(* CoDeSys 2.3.9.1 project: oscat270.pro *)
(* Libraries: SysLibSockets.lib 14.4.05 11:11:38, WagoLibEthernet_01.lib 9.8.07 10:37:24, SysLibRtc.lib 5.10.04 09:37:42, Standard.lib 22.11.04 11:21:12, SYSLIBCALLBACK.LIB 20.4.05 10:04:48 *)

(* Global variable list: Constants *)
VAR_GLOBAL CONSTANT
	(* setup Parameters *)
	STEP7 : BOOL := FALSE;

	(* Mathematische Konstanten *)
	PI1 : REAL := 3.14159265358979323846264338327950288;	(* Kreiszahl PI *)
	PI2 : REAL := 6.283185307179586476;					(* PI * 2 *)
	E : REAL := 2.71828182845904523536028747135266249;	(* Eulersche Konstante *)

	(* Physikalische Konstanten *)
	C0 : REAL := 299792458 ;							(* Lichtgeschwindigkeit in m/s *)
	EL : REAL := 1.60217653E-19;						(* elementarladung in Colomb = A * s *)
	GN : REAL := 9.80665; 								(* Erdbeschleunigung in m / s² *)
	TK : REAL := -273.15;									(* absoluter Nullpunkt in °C *)
	RU : REAL := 8.314472; 								(*Universelle Gaskonstante in J / (mol · K) *)
	PN : REAL := 101325;									(* NormalDruck in Pa *)

END_VAR

VAR_GLOBAL
END_VAR

(* revisionhistory
hm 3.3.2007
	extended accuracy of pi2
	renamed T0 to Tk for better compatibility with other libraries
	renamed C t0 c0 for better compatibility

hm	2.5.2007
	added RU universal gas constant

hm	1. oct 2007
	added setup parameter STEP7

hm 31. oct 2007
	added PN
*)

(* Data type *)
TYPE esr_data :
STRUCT
	typ : BYTE;
	adress : STRING(10);
	DS : DT;
	TS : TIME;
	data : ARRAY[0..7] OF BYTE;
END_STRUCT
END_TYPE

(* Data type *)
TYPE vector_3 :
STRUCT
	X : REAL;
	Y : REAL;
	Z : REAL;
END_STRUCT
END_TYPE

(* POU XTEST/PLC_PRG, CFC *)
PROGRAM PLC_PRG
VAR
END_VAR
VAR_INPUT
END_VAR
_CFC_ (* Continuous Function Chart, elements in execution order *)
_END_CFC_
END_PROGRAM

(* POU XTEST/Baustein Tests/air_test, CFC *)
PROGRAM air_test
VAR
	temp: REAL := 70;
	den: REAL;
	den1: REAL;
	ent: REAL;
	cp: REAL;
	rh: REAL := 0.5;
	P: REAL := 101325;
	ice: BOOL;
	SDx: REAL;
	enth: REAL;
END_VAR
VAR (* helpers for the ST form of the networks *)
	_t1 : REAL;
	_t58 : REAL;
END_VAR
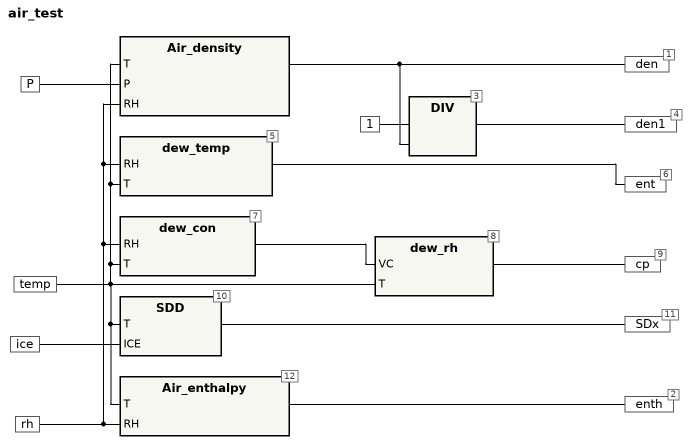
_CFC_ (* Continuous Function Chart, elements in execution order *)
#0 Air_density(T: temp, P: P, RH: rh)
#1 den <= #0
#2 enth <= #12
#3 DIV(1, #0)
#4 den1 <= #3
#5 dew_temp(RH: rh, T: temp)
#6 ent <= #5
#7 dew_con(RH: rh, T: temp)
#8 dew_rh(VC: #7, T: temp)
#9 cp <= #8
#10 SDD(T: temp, ICE: ice)
#11 SDx <= #10
#12 Air_enthalpy(T: temp, RH: rh)
_END_CFC_
(* the same logic as Structured Text *)
_t1 := Air_density(T := temp, P := P, RH := rh);
den := _t1;
enth := _t58;
den1 := 1 / _t1;
ent := dew_temp(RH := rh, T := temp);
cp := dew_rh(VC := dew_con(RH := rh, T := temp), T := temp);
SDx := SDD(T := temp, ICE := ice);
_t58 := Air_enthalpy(T := temp, RH := rh);
END_PROGRAM

(* POU mathematical/neg, ST *)
FUNCTION neg : INT
VAR_INPUT
	in : INT;
END_VAR
VAR
	X : WORD := 2#1111_1111_1111_1111;
END_VAR

(*
version 1.0	11 nov 2007
programmer 	hugo
tested by		tobias

this function return the value of in multiplied by -1

*)
neg := WORD_TO_INT(INT_TO_WORD(in - 1) XOR X);

(* revision history
hm 11.11.2007	rev 1.0
	original version

*)
END_FUNCTION

(* POU Building/HLK/Air_density, ST *)
FUNCTION Air_density : REAL
VAR_INPUT
	T : REAL;
	P : REAL;
	RH : REAL;
END_VAR
VAR CONSTANT
	RL : REAL := 287.05;
	RX : REAL := 3.773319E-3;
END_VAR
VAR
END_VAR

(*
version 1.1	4 dec 2007
programmer 	hugo
tested by		tobias

this function calculates the air density between 0 and 100 deg C

*)
Air_density := PN * (1 - RH * SDD(T, TRUE) * RX / P) / (RL * ( T - TK));

(* original code used for rev 1.0

SDD := SDD(T,FALSE);
RF := RL / (1- RH*SDD/P*RX);
Air_density := P / (RF * (T-TK));

*)

(* revision history

hm	29.10.2007		rev 1.0
	original version

hm	4.12.2007		rev 1.1
	changed code for better performance

*)
END_FUNCTION

(* POU Building/HLK/SDD, ST *)
FUNCTION SDD : REAL
VAR_INPUT
	T : REAL;
	ICE: BOOL;
END_VAR
VAR CONSTANT
END_VAR
VAR
END_VAR

(*
version 1.1	2 dec 2007
programmer 	hugo
tested by		tobias

this function calculates the vapor saturation pressure for moist Air over ice or water

*)
IF ice THEN
	SDD := 611.153 * EXP(22.4433 * T / (272.186 + T));
ELSE
	SDD := 611.213 * EXP(17.5043 * T / (241.2 + T));
END_IF;

(* old code used in rev 1.0
IF ice THEN
	SDD := 611.153 * exp10(9.747*T / (272.186 + T));
ELSE
	SDD := 611.213 * exp10(7.602*T / (241.2 + T));
END_IF;
*)


(* revision history

hm 29 oct 2007		rev 1.0
	original version

hm	2. dec 2007		rev 1.1
	changed code for better performance
*)
END_FUNCTION

(* POU Building/HLK/dew_temp, ST *)
FUNCTION dew_temp : REAL
VAR_INPUT
	RH : REAL;
	T : REAL;
END_VAR
VAR CONSTANT
	a : REAL := 7.5;
	b : REAL := 237.3;
END_VAR
VAR
	V : REAL;
END_VAR

(*
version 1.4	8 jan 2008
programmer 	hugo
tested by		tobias

this function calculates the dew point for air given the temperature and relative humidity.
dew_temp(60,0.25) = 16.7 °C.
which means the dew point for air with 25° and 60% RH is at 16.7 °C.


*)
IF rh > 0 THEN
(*	old code was rewritten for better performance
	SDD := 6.1078*EXPT(10,(a*T)/(b+T));
	DD := RH/100 * SDD;
	V := LOG(DD/6.1078);
	dew_temp := b*V/(a-v);
*)
	V := LOG(RH * 0.01 * exp10((a*T)/(b+T)));
	dew_temp := b*V/(a-V);
ELSE
	dew_temp:= -TK;
END_IF;

(* revision history

hm		2.10.2006	rev 1.0
	original version created

hm		29.4.2007	rev 1.1
	checked for rh not to be 0 because log(0) is not defined

hm		13.9.2007	rev 1.2
	code rewritten for better performance

hm		2. dec 2007	rev 1.3
	changed code for better performance

hm		8. jan 2008	rev 1.4
	further improvement in performance
*)

(*
Bezeichnungen:
r = relative Luftfeuchte
T = Temperatur in °C
TK = Temperatur in Kelvin (TK = T + 273.15)
TD = Taupunkttemperatur in °C
DD = Dampfdruck in hPa
SDD = Sättigungsdampfdruck in hPa

Parameter:
a = 7.5, b = 237.3 für T >= 0
a = 7.6, b = 240.7 für T < 0 über Wasser (Taupunkt)
a = 9.5, b = 265.5 für T < 0 über Eis (Frostpunkt)

R* = 8314.3 J/(kmol*K) (universelle Gaskonstante)
mw = 18.016 kg (Molekulargewicht des Wasserdampfes)
AF = absolute Feuchte in g Wasserdampf pro m3 Luft

Formeln:

   1. SDD(T) = 6.1078 * 10^((a*T)/(b+T))
   2. DD(r,T) = r/100 * SDD(T)
   3. r(T,TD) = 100 * SDD(TD) / SDD(T)
   4. TD(r,T) = b*v/(a-v) mit v(r,T) = log10(DD(r,T)/6.1078)
   5. AF(r,TK) = 10^5 * mw/R* * DD(r,T)/TK; AF(TD,TK) = 10^5 * mw/R* * SDD(TD)/TK 

*)
END_FUNCTION

(* POU mathematical/exp10, ST *)
FUNCTION exp10 : REAL
VAR_INPUT
	X : REAL;
END_VAR
VAR
END_VAR

(*
version 1.0	 2 dec 2007
programmer 	hugo
tested by		tobias

this function calculates the exponent to the basis 10
exp10(3) = 1000

*)
exp10 := EXP(X * 2.30258509299405);

(* revision history
hm	2. dec 2007		rev 1.0
	original version

*)
END_FUNCTION

(* POU Building/HLK/dew_con, ST *)
FUNCTION dew_con : REAL
VAR_INPUT
	RH : REAL;
	T : REAL;
END_VAR
VAR CONSTANT
END_VAR
VAR
END_VAR

(*
version 1.2	2 dec 2007
programmer 	hugo
tested by		tobias

this function calculates the water concentratin in air for a given temperature and relative humidity.
the output states the concentration of water vapor in air in Gramms / qubic meter.

*)
IF rh > 0 THEN
(*	this code is good to read but need to be improoved
	SDD := 6.1078*EXPT(10,(a*T)/(b+T));
	DD := RH/100 * SDD;
	V := LOG(DD/6.1078);
	TD := b*V/(a-v);
	dew_con := 0.1 * mw / RU * DD / (T - TK);
*)
	dew_con := 2.166824303E-2 * RH * SDD(T,FALSE)  / (T - TK);
ELSE
	dew_con := 0;
END_IF;

(*
Bezeichnungen:
r = relative Luftfeuchte
T = Temperatur in °C
TK = Temperatur in Kelvin (TK = T + 273.15)
TD = Taupunkttemperatur in °C
DD = Dampfdruck in hPa
SDD = Sättigungsdampfdruck in hPa

Parameter:
a = 7.5, b = 237.3 für T >= 0
a = 7.6, b = 240.7 für T < 0 über Wasser (Taupunkt)
a = 9.5, b = 265.5 für T < 0 über Eis (Frostpunkt)

R* = 8314.3 J/(kmol*K) (universelle Gaskonstante)
mw = 18.016 kg (Molekulargewicht des Wasserdampfes)
AF = absolute Feuchte in g Wasserdampf pro m3 Luft

Formeln:

   1. SDD(T) = 6.1078 * 10^((a*T)/(b+T))
   2. DD(r,T) = r/100 * SDD(T)
   3. r(T,TD) = 100 * SDD(TD) / SDD(T)
   4. TD(r,T) = b*v/(a-v) mit v(r,T) = log10(DD(r,T)/6.1078)
   5. AF(r,TK) = 10^5 * mw/R* * DD(r,T)/TK; AF(TD,TK) = 10^5 * mw/R* * SDD(TD)/TK 

*)

(* revision history

hm 29 apr 2007		rev 1.0
	original version

hm	13.sep 2007		rev 1.1
	improoved coding for speed
	deleted unused variabled SDD,DD,V, TD

hm	2. dec 2007		rev 1.2
	changed code for better performance
	output is now in Gramms / Qubic meter
*)
END_FUNCTION

(* POU Building/HLK/dew_rh, ST *)
FUNCTION dew_rh : REAL
VAR_INPUT
	VC : REAL;
	T : REAL;
END_VAR

(*
version 1.1	2 dec 2007
programmer 	hugo
tested by		tobias

this function calculates the relative humidity in air for a given temperature in °C and vapor concentration in Kg/m³..

*)
dew_rh := LIMIT(0,VC / dew_con(1,T),100);

(* code before rev 1.1
dew_rh := VC / dew_con(100,T) * 100;
IF dew_rh > 100 THEN dew_rh := 100; END_IF;
*)

(* revision history
hm		29. apr 2007	rev 1.0
	original version

hm		2. 12. 2007		rev 1.1
	new code for better performance

*)
END_FUNCTION

(* POU Building/HLK/Air_enthalpy, ST *)
FUNCTION Air_enthalpy : REAL
VAR_INPUT
	T : REAL;
	RH : REAL;
END_VAR
VAR CONSTANT
	CPL : REAL := 1.00482;
	CW : REAL := 1.86;
	LH : REAL := 2500.78;
END_VAR
VAR
END_VAR

(*
version 1.1	2 nov 2007
programmer 	hugo
tested by		tobias

this function calculates the enthalpy for humid air between 0 and 100 deg C

*)
Air_enthalpy := CPL * T + (CW * T + LH) * dew_con(RH,T);

(* revision history

hm	31.10.2007		rev 1.0
	original version

hm	2.11.2007		rev 1.1
	deleted unused variable RF

hm	2.12.2007		rev 1.2
	changed code for better performance
*)
END_FUNCTION

(* POU XTEST/Baustein Tests/bcd_test, CFC *)
PROGRAM bcd_test
VAR
	strbcd: STRING;
	inout: INT;
	inx: INT;
END_VAR
VAR_INPUT

END_VAR
VAR (* helpers for the ST form of the networks *)
	_t16 : BCD;
	_t15 : INT;
END_VAR
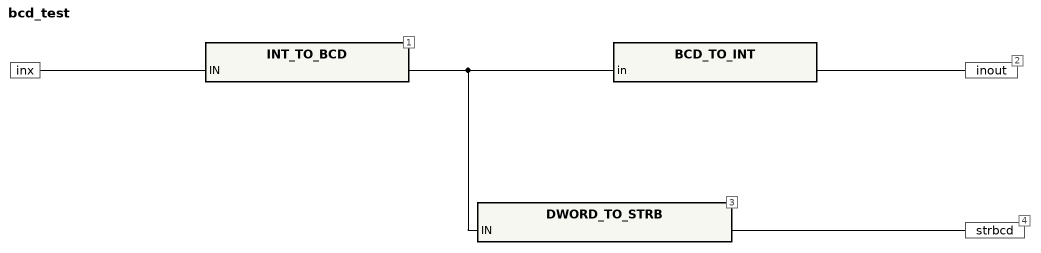
_CFC_ (* Continuous Function Chart, elements in execution order *)
#0 BCD_TO_INT(in: #1)
#1 INT_TO_BCD(IN: inx)
#2 inout <= #0
#3 DWORD_TO_STRB(IN: #1)
#4 strbcd <= #3
_END_CFC_
(* the same logic as Structured Text *)
_t15 := BCD_TO_INT(in := _t16);
_t16 := INT_TO_BCD(IN := inx);
inout := _t15;
strbcd := DWORD_TO_STRB(IN := _t16);
END_PROGRAM

(* POU Logic/gate logic/BCD_TO_INT, ST *)
FUNCTION BCD_TO_INT : INT
VAR_INPUT
	in : BYTE;
END_VAR
VAR
END_VAR

(*
version 1.0	13 dec 2007
programmer 	hugo
tested by		tobias

this function converts a two digit bcd number into an integer.
*)
	BCD_TO_INT := (in AND 16#0F) + (SHR(in,4) * 10);

(* revision history
hm	13.12.2007
	original version

*)
END_FUNCTION

(* POU Logic/gate logic/INT_TO_BCD, ST *)
FUNCTION INT_TO_BCD : BYTE
VAR_INPUT
	IN : INT;
END_VAR
VAR
END_VAR

(*
version 1.0	17 jan 2007
programmer 	hugo
tested by		tobias

this function converts an integer into a two digit bcd number.
*)
INT_TO_BCD := INT_TO_BYTE(SHL(TRUNC(in/10),4) + (in MOD 10));

(* revision history
hm	13.12.2007
	original version

*)
END_FUNCTION

(* POU String/DWORD_TO_STRB, ST *)
FUNCTION DWORD_TO_STRB : STRING
VAR_INPUT
	IN : DWORD;
END_VAR
VAR
	pt : POINTER TO BYTE;
	i: INT;
END_VAR

(*
version 1.1	15 dec 2007
programmer 	hugo
tested by		tobias

DWORD_TO_STRINGB converts a DWORD to a String of Bits represented by '0' and '1' s.
The lowest order bit will be on the right and the high order bit on the left.

*)
(* pointer für die ausgabe ermitteln *)
pt := ADR(DWORD_TO_STRB);
(* die 8 ausgabecharacter ermitteln und schreiben *)
FOR i := 1 TO 32 DO
	IF in.31 THEN pt^ := 49; ELSE pt^ := 48; END_IF;
	in := SHL(in,1);
	pt := pt + 1;
END_FOR;

(* der ausgabestring muss nochg mit 0 abgeschlossen werden *)
pt^ := 0;

(* revision history
hm		9.6.2007	rev 1.0		
	original version 
hm		15.dec 2007	rev 1.1
	changed code for better performance
*)
END_FUNCTION

(* POU XTEST/Baustein Tests/blind_test, CFC *)
PROGRAM blind_test
VAR
	up: BOOL;
	dn: BOOL;
	x1: blind_scene;
	mu: BOOL;
	md: BOOL;
	pos: BYTE;
	ang: BYTE;
	x2: blind_security;
	esr: BYTE;
	fire: BOOL;
	wind: BOOL;
	alarm: BOOL;
	rain: BOOL;
	x3: blind_control;
	x5: blind_input;
	p: BYTE;
	a: BYTE;
	IN: BOOL;
	utc: DT;
	X7: blind_night;
	x8: sun_time;
	Door: BOOL;
	x9: sun_pos;
	x10: BLIND_SHADE;
	S_write: BOOL;
	S_enable: BOOL;
	scene: BYTE;
	sun: BOOL;
	ex: BOOL;
END_VAR
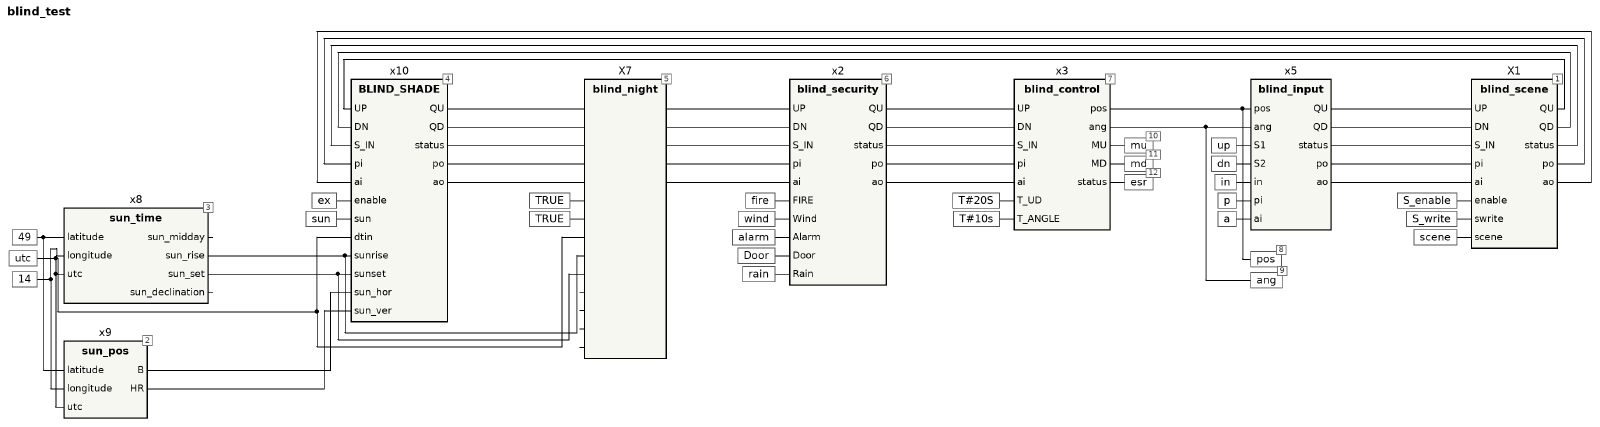
_CFC_ (* Continuous Function Chart, elements in execution order *)
#0 x5:blind_input(pos: #7.pos, ang: #7.ang, S1: up, S2: dn, in: in, pi: p, ai: a, click_mode := TRUE, click_time := T#250ms, manual_timeout := T#10s)
#1 X1:blind_scene(UP: #0.QU, DN: #0.QD, S_IN: #0.status, pi: #0.po, ai: #0.ao, enable: S_enable, swrite: S_write, scene: scene)
#2 x9:sun_pos(latitude: 49, longitude: 14, utc: utc)
#3 x8:sun_time(latitude: 49, longitude: 14, utc: utc)
#4 x10:BLIND_SHADE(UP: #1.QU, DN: #1.QD, S_IN: #1.status, pi: #1.po, ai: #1.ao, enable: ex, sun: sun, dtin: utc, sunrise: #3.sun_rise, sunset: #3.sun_set, sun_hor: #2.B, sun_ver: #2.HR, direction := 180, slat_width := 60, Slat_spacing := 60)
#5 X7:blind_night(#4.QU, #4.QD, #4.status, #4.po, #4.ao, TRUE, TRUE, utc, #3.sun_rise, #3.sun_set, -, -, -, -)
#6 x2:blind_security(UP: #5.out 1, DN: #5.out 2, S_IN: #5.out 3, pi: #5.out 4, ai: #5.out 5, FIRE: fire, Wind: wind, Alarm: alarm, Door: Door, Rain: rain, Alarm_UP := TRUE)
#7 x3:blind_control(UP: #6.QU, DN: #6.QD, S_IN: #6.status, pi: #6.po, ai: #6.ao, T_UD: T#20S, T_ANGLE: T#10s, sens := 5, T_Lockout := T#3s)
#8 pos <= #7.pos
#9 ang <= #7.ang
#10 mu <= #7.MU
#11 md <= #7.MD
#12 esr <= #7.status
_END_CFC_
END_PROGRAM

(* POU Building/Jalousie/blind_scene, ST *)
FUNCTION_BLOCK blind_scene
VAR_INPUT
	UP, DN : BOOL;
	S_IN : BYTE;
	pi, ai : BYTE;
	enable : BOOL;
	swrite : BOOL;
	scene : BYTE;
END_VAR
VAR_INPUT CONSTANT
END_VAR
VAR_OUTPUT
	QU, QD : BOOL;
	status : BYTE;
	po, ao : BYTE;
END_VAR
VAR RETAIN
	sx : ARRAY[0..15,0..2] OF BYTE;
END_VAR
VAR_TEMP
	x : BYTE;

END_VAR

(*
version 1.1	29. jan 2008
programmer 	hugo
tested by		tobias


*)
(* delete all bits except the lower 4 of scene *)
x := scene AND 16#0F;

IF enable AND sx[x,2] > 0 AND UP AND DN THEN
	po := sx[x,0];
	ao := sx[x,1];
	status := 160 + x;  (* Status number is 160 to 175 for the 16 scenes *)
	QU := TRUE;
	QD := TRUE;
ELSE
	QU := UP;
	QD := DN;
	status := S_IN;
	po := pi;
	ao := ai;
END_IF;

(* write scene if necessary *)
IF swrite THEN
	status := 176;		(* write scene *)
	sx[x,0] := pi;
	sx[x,1] := ai;
	IF enable THEN sx[x,2] := 1; ELSE sx[x,2] := 0; END_IF; (* if sx[x,2] = 0 the scene is disabled *)
END_IF;


(* revision history
hm	24. oct 2007	rev 1.0
	original release

hm		29.1.2008	rev 1.1
	replaced shr/shl with and for better performance
*)
END_FUNCTION_BLOCK

(* POU Building/Jalousie/blind_security, ST *)
FUNCTION_BLOCK blind_security
VAR_INPUT
	UP, DN : BOOL;
	S_IN : BYTE;
	pi, ai : BYTE;
	FIRE : BOOL;
	Wind : BOOL;
	Alarm : BOOL;
	Door : BOOL;
	Rain : BOOL;
END_VAR
VAR_INPUT CONSTANT
	Alarm_UP : BOOL := TRUE;
END_VAR
VAR_OUTPUT
	QU, QD : BOOL;
	status : BYTE;
	po, ao : BYTE;
END_VAR
VAR
END_VAR

(*
version 1.1	6. oct 2007
programmer 	hugo
tested by		tobias


*)
IF Fire THEN
	QU := TRUE;
	QD := FALSE;
	status := 111;
ELSIF Wind THEN
	QU := TRUE;
	QD := FALSE;
	status := 112;
ELSIF alarm THEN
	QU := Alarm_up;
	QD := NOT Alarm_up;
	status := 113;
ELSIF Door THEN
	QU := TRUE;
	QD := FALSE;
	status := 114;
ELSIF Rain AND NOT (up XOR dn) THEN
	QU := FALSE;
	QD := TRUE;
	status := 115;
ELSE
	QU := UP;
	QD := DN;
	status := S_IN;
	po := pi;
	ao := ai;
END_IF;


(* revision history
hm	29. sep 2007	rev 1.0
	original release

hm	6. oct 2007		rev 1.1
	added pos and angle inputs and outputs
	manual will override rain position
	alarm position can now be configured

*)
END_FUNCTION_BLOCK

(* POU Building/Jalousie/blind_control, ST *)
FUNCTION_BLOCK blind_control
VAR_INPUT
	UP, DN : BOOL;
	S_IN : BYTE;
	pi : BYTE;
	ai : BYTE;
	T_UD, T_ANGLE : TIME;
END_VAR
VAR_INPUT CONSTANT
	sens : BYTE := 5;
	T_Lockout: TIME := T#100ms;
END_VAR
VAR_OUTPUT
	pos, ang : BYTE;
	MU, MD : BOOL;
	status : BYTE;
END_VAR
VAR
	act : blind_actuator;
	delta : BYTE;
END_VAR

(*
version 1.3	30. oct 2007
programmer 	hugo
tested by		tobias


*)
IF UP AND DN THEN
	(* automatic modus detected *)
	(* first find correct position *)
	IF BYTE_TO_INT(act.pos) < BYTE_TO_INT(pi) - delta THEN
		act.UP := TRUE;
		act.DN := FALSE;
		delta := 0;
		act.S_IN := 121;
	ELSIF BYTE_TO_INT(act.pos) > BYTE_TO_INT(pi) + delta THEN
		act.UP := FALSE;
		act.DN := TRUE;
		delta := 0;
		act.S_IN := 122;
	(* regulate angle *)
	ELSIF BYTE_TO_INT(act.ang) < BYTE_TO_INT(ai) - delta AND T_angle > T#100ms THEN
		act.UP := TRUE;
		act.DN := FALSE;
		delta := 0;
		act.S_IN := 123;
	ELSIF BYTE_TO_INT(act.ang) > BYTE_TO_INT(ai) + delta AND T_angle > T#100ms THEN
		act.UP := FALSE;
		act.DN := TRUE;
		delta := 0;
		act.S_IN := 124;
	(* correct position reached *)
	ELSE
		act.UP := FALSE;
		act.DN := FALSE;
		delta := sens;
		act.S_IN := 0;
	END_IF;
ELSE
	act.UP := UP;
	act.DN := DN;
END_IF;

(* hand over status *)
IF s_in > 0 THEN act.S_IN := S_IN; END_IF;

(* blind control calls blind_actuator *)
act(T_UD:=T_UD, T_ANGLE:=T_ANGLE, T_lockout := T_Lockout);
pos := act.pos;
ang := act.ang;
MU := act.QU;
md := act.QD;
status := act.status;

(* revision history
hm	29. sep 2007	rev 1.0
	original release

hm	6. oct 2007		rev 1.1
	rearranged outputs
	integrated blind_actuator into blind_control

hm	16. oct 2007	rev 1.2
	ignore angle when t_angle = 0

hm 29. oct 2007	rev 1.3
	added lockout configuration time for motor direction change
	sens has a setup value of 5
*)
END_FUNCTION_BLOCK

(* POU Building/Jalousie/blind_actuator, ST *)
 FUNCTION_BLOCK blind_actuator
VAR_INPUT
	UP, DN : BOOL;
	S_IN : BYTE;
	T_UD : TIME := T#10s;
	T_Angle : TIME := T#3s;
END_VAR
VAR_INPUT CONSTANT
	T_lockout : TIME := t#100ms;
END_VAR
VAR_OUTPUT
	pos, ang : BYTE;
	QU, QD : BOOL;
	status : BYTE;
END_VAR
VAR
	position, angle : rmp_B;
	lock : interlock;
END_VAR

(*
version 1.1	6 oct 2007
programmer 	hugo
tested by		tobias

blind actuator drives the up and down motor of a blind. T_lockout specifies the time between up or dn becomes active. 
To change direction there must be a minimum wait time to allow the motors to come to rest first.
the up and down outputs QU and QD are controlled by the inputs UP and DN.
the outputs pos and ang simulate the position of the blind pos = 0 means blind is down and pos = 255 = blind is up.
the angle 0 means vertical posisition of the slates and 255 means horizontal position of the slates.


*)
(* make sure only one motor is active at a given time *)
lock(i1 := UP, I2 := DN, TL := T_lockout);

(* ramp up or down to simulate the angle position of the blind slats *)
angle(en := lock.Q1 OR lock.Q2, UP := lock.Q1, PT := T_Angle);
position(en := lock.Q1 AND angle.high OR lock.Q2 AND angle.low, up := lock.Q1, PT := T_UD);

(* set the outputs *)
pos := position.Out;
ang := angle.Out;
QU := lock.Q1;
QD := lock.Q2;

(* set the status output *)
IF UP AND DN THEN
	IF s_in < 10 AND S_in > 1 THEN status := s_in; ELSE status := 1; END_IF;			(* error up and down together are not allowed *)
ELSIF S_IN > 0 THEN
	status := S_IN;
ELSIF UP THEN
	status := 101;
ELSIF DN THEN
	status := 102;
ELSE
	status := 0;
END_IF;


(* revision history
hm	29. sep 2007	rev 1.0
	original release

hm	6. oct 2007		rev 1.1
	rearranged outputs
	
*)
END_FUNCTION_BLOCK

(* POU engineering/signal generators/rmp_B, ST *)
FUNCTION_BLOCK rmp_B
VAR_INPUT
	SET : BOOL := FALSE;
	PT : TIME;
	EN : BOOL := TRUE;
	UP : BOOL := TRUE;
	RST : BOOL := FALSE;
END_VAR
VAR_OUTPUT
	out : BYTE;
	busy: BOOL;
	high : BOOL;
	low : BOOL;
END_VAR
VAR
	last_step : DWORD;
	now : DWORD;
	tmp: DWORD;
	edge: BOOL;
	N : BYTE;
	init: BOOL;
END_VAR

(*
	version 1.6	25 dec 2007
	programmer 	oscat
	tested BY		oscat

this ramp generator generates a byte wide ramp with 255 steps
the generator has an asynchronous set and reset
the ramp is controlled by PT which is the total ramp time for a full sweep from 0..255
an UD input controlls the direction Up or Down and the E input enables the ramp generation
a busy output indicates that the ramp is running, busy false means output is stable.
the outputs low and high will be true when the output has reached its max or min value.

*)
(* read system time *)
now := T_PLC_MS();

(* init code for startup *)
IF NOT init THEN
	init := TRUE;
	last_step := now;
END_IF;

(* calculate the necessary step response *)
IF pt = t#0s THEN
	tmp := 255;
ELSE
	tmp := SHL(now - last_step, 8) / (TIME_TO_DWORD(pt));
END_IF;
IF tmp > 255 THEN N:= 255; ELSE N:= DWORD_TO_BYTE(tmp); END_IF;

(* detetct edge on en *)
IF en AND NOT edge THEN
	last_step := now;
(* check for asynchronous set or reset *)
ELSIF rst THEN
	out := 0;
ELSIF set  THEN
	out := 255;
ELSIF en AND N > 0 THEN
	(* generate ramp *)
	last_step := now;
	IF UP THEN
		IF out > 255 - N THEN out := 255; ELSE out := out + N; END_IF;
	ELSE
		IF out < N THEN out := 0; ELSE out := out - N; END_IF;
	END_IF;
END_IF;
edge := en;

(* checks for outputs stable and reset or set busy flag *)
IF out = 0 THEN
	busy := FALSE;
	low := TRUE;
	high := FALSE;
ELSIF out = 255 THEN
	busy := FALSE;
	high := TRUE;
	low := FALSE;
ELSE
	busy := en;
	high := FALSE;
	low := FALSE;
END_IF;


(* revision history

hm 5.10.2006	rev 1.1
	added busy output
hm 17.1.2007	rev 1.2
	renamed input ud to up for better usability
	deleted unused variable step

hm	17.9.2007	rev 1.3
	replaced time() with t_plc_ms() for compatibility reasons

hm	28. sep 2007	rev 1.4
	added outputs on and off
	busy is now disabled while en is false
	new coding for higher accuracy and performance

hm	5. oct 2007		rev 1.5
	added statements to allow for PT to be t#0s output jumps to max or min immediately

hm	25. dec 2007	REV 1.6
	IMPROOVED CODE FOR BETTER PERFORMANCE
*)
END_FUNCTION_BLOCK

(* POU engineering/measurements/T_PLC_MS, ST *)
FUNCTION T_PLC_MS : DWORD
VAR CONSTANT
	debug : BOOL := FALSE;
	N : INT := 0;
	offset : DWORD := 0;
END_VAR
VAR
	tx : TIME;
	temp : DWORD := 1;
END_VAR

(*
version 1.1	12 nov 2007
programmer 	hugo
tested by		tobias

T_PLC_MS reads the internal PLC timer and return the time, it has the advantage to be able to set a debug mode 
and speed up the counter to test the plc timer overrun which occurs every 50 days respectively 25 days at siemens S7
this routine also allows to correct the behavior of s7 where the internal plc counter will not count all 32 bits.

*)
tx := TIME();
T_PLC_MS := TIME_TO_DWORD(Tx);
(* hier muss die korrektur für step7 stattfinden
plctime muss den vollen wertebereich von time ausnutzen:
wenn bei step7 time -24tage bis plus 24 tage ist dann muss der timer auch beim überlauf auf -24tage springen 
und auf keinen fall auf 0 !!!!
für siemens muss ein weiterer fb im main eingebunden werden der sicherstellt das alle 32 bits durchgezählt werden.
es kann nur ein fb sein den er muss sich das oberste (32te) bit merken.
oder etwa spring s7 bei überlauf auf -24 tage????? dann wäre keine korrektur nötig.
*)
IF debug THEN
	T_PLC_MS := (SHL(T_PLC_MS,N) OR SHL(temp,N)-1) + Offset;
END_IF;

(* revision history
hm	14.9.2007	rev 1.0
	original version

hm	12. nov 2007	rev 1.1
	added temporaray variable tx because some compilers could not handle time() as an argument

*)
END_FUNCTION

(* POU engineering/signal processing/Offset, ST *)
FUNCTION Offset : REAL
VAR_INPUT
	X : REAL;
	O1, O2, O3, O4 : BOOL;
	D : BOOL;
END_VAR
VAR_INPUT CONSTANT
	Offset_1 : REAL;
	Offset_2 : REAL;
	Offset_3 : REAL;
	Offset_4 : REAL;
	default : REAL;
END_VAR

(*
version 1.0	12 jan 2007
programmer 	oscat
tested by		tobias

The Function offset adds offsets to an analog signal depending on digital inputs.
all selected offsets are added at the same time.
with the input D a default value instead of the input X can be used.

*) 
IF D THEN Offset := default; ELSE Offset := X; END_IF;
IF O1 THEN Offset := Offset + offset_1; END_IF;
IF O2 THEN Offset := Offset + offset_2; END_IF;
IF O3 THEN Offset := Offset + offset_3; END_IF;
IF O4 THEN Offset := Offset + offset_4; END_IF;
END_FUNCTION

(* POU engineering/automation/interlock, ST *)
FUNCTION_BLOCK interlock
VAR_INPUT
	I1, I2 : BOOL;
	TL : TIME;
END_VAR
VAR_OUTPUT
	Q1, Q2 : BOOL;
END_VAR
VAR
	T1, T2 : TOF;
END_VAR

(*
version 1.0	28 sep 2007
programmer 	hugo
tested by		tobias

INTERLOCK has two inputs I1 and I2 which drive the corresponding outputs Q1 and Q2.
the inputs signals lock each other out and therfore I1 can only drive Q1 when I2 is Low and vice versa.
The input TL specifies a dead time between two outputs can become active.
an output can only become active when the other output was not active for the time TL.

*)
(* the input signal have a run delay to lockout the other input *)
T1(IN := I1, PT := TL);
T2(IN := I2, PT := TL);

Q1 := I1 AND NOT t2.Q;
Q2 := I2 AND NOT t1.Q;


(* revision history

hm	28 sep 2007		rev 1.0
	original version

*)
END_FUNCTION_BLOCK

(* POU Building/Jalousie/blind_input, ST *)
FUNCTION_BLOCK blind_input
VAR_INPUT
	pos, ang : BYTE;
	S1, S2 : BOOL;
	in : BOOL;
	pi, ai : BYTE;
END_VAR
VAR_INPUT CONSTANT
	single_switch : BOOL := FALSE;
	click_mode : BOOL := TRUE;
	click_time : TIME := T#200ms;
	click_timeout : TIME := T#60s;
	manual_timeout: TIME := T#1h;
END_VAR
VAR_OUTPUT
	QU, QD : BOOL;
	status : BYTE;
	po, ao : BYTE;
END_VAR
VAR
	click_run : TOF;
	tog1, tog2 : TOGGLE;
	pl1, pl2 : Pulse_Length;
	SU, SD : BOOL;
	last_act: DWORD;
	tx: DWORD;
END_VAR

(*
version 1.2	30 dec 2007
programmer 	hugo
tested by		tobias


*)
(* read system_time *)
tx := T_PLC_MS();

(* single or double switch operation *)
IF click_mode THEN
	PL1(in := S1, T_short := click_time, T_long := click_time);
	PL2(in := S2, T_short := click_time, T_long := click_time);
	(* a timeout needs to be added for click enable *)
	click_run(IN := pl1.short OR pl2.short, PT := click_timeout);
	tog1(clk := pl1.short, rst := pl1.long OR pl2.short OR pl2.long OR NOT click_run.Q);
	tog2(clk := pl2.short, rst := pl2.long OR pl1.short OR pl1.long OR NOT click_run.Q);

	SU := tog1.Q OR PL1.long;
	SD := tog2.Q OR pl2.long;
ELSE
	tog1(CLK := NOT S1);
	SU := (S1 AND NOT tog1.Q AND single_switch) OR (NOT single_switch AND S1);
	SD := (S1 AND tog1.Q AND single_switch) OR (NOT single_switch AND S2);
END_IF;

(* Forced Input is active *)
IF in THEN
	QU := TRUE;
	QD := TRUE;
	po := pi;
	ao := ai;
	status := 131;

(* in manual mode set ps and as to actual values *)
ELSIF SU OR SD THEN
	po := pos;
	ao := ang;
	last_act := tx;
	QU := SU;
	QD := SD;
	IF su THEN status := 132; ELSE status := 133; END_IF;

(* enable automatik mode after auto timer has expired *)
ELSIF manual_timeout > t#0s AND tx - last_act >= TIME_TO_DWORD(manual_timeout) THEN
	QU := TRUE;
	QD := TRUE;
	status := 134;

(* no input active *)
ELSE
	QU := FALSE;
	QD := FALSE;
	status := 0;
END_IF;


(* revision history
hm	29. sep 2007	rev 1.0
	original release

hm	6. oct 2007		rev 1.1
	renamed ps and as to po and ao

hm	30. dec 2007	rev 1.2
	added click_timeout variable and function

*)
END_FUNCTION_BLOCK

(* POU Logic/FF edge triggered/TOGGLE, ST *)
FUNCTION_BLOCK TOGGLE
VAR_INPUT
	CLK : BOOL;
	rst : BOOL := FALSE;
END_VAR
VAR_OUTPUT
	Q : BOOL;
END_VAR
VAR
	edge : BOOL;
END_VAR

(*
version 1.0	13 sep 2007
programmer 	hugo
tested by		tobias

toggle flip flop the output changes state with every rising edge of clk.

*)
IF rst THEN
	q := 0;
ELSIF clk AND NOT edge THEN
	Q := NOT Q;
END_IF;
edge := clk;

(* revision history

hm	13.9.2007		rev 1.0
	original version

*)
END_FUNCTION_BLOCK

(* POU Building/electrical/Pulse_Length, ST *)
FUNCTION_BLOCK Pulse_Length
VAR_INPUT
	in : BOOL;
END_VAR
VAR_OUTPUT
	short : BOOL;
	middle : BOOL;
	long : BOOL;
END_VAR
VAR_INPUT CONSTANT
	T_short : TIME := t#100ms;
	T_long : TIME := t#1s;
END_VAR
VAR
	tx : TIME;
	tn: TIME;
	edge : BOOL;
END_VAR

(*
version 1.1	15 sep 2007
programmer 	oscat
tested by		tobias

Pulse_length indicates on 3 outputs if an input pulse had been shorter than T_short (short = True), longer than T_long (long = True) or between T_short and T_long (middle = True).

*)
(* read system time *)
tx := DWORD_TO_TIME(T_PLC_MS());

(* reset outputs, they should only be active 1 cycle *)
short := FALSE;
Middle := FALSE;
long := FALSE;

(* detect rising edge *)
IF in AND NOT edge THEN
	edge := TRUE;
	tn := tx;

(* detect for falling edge *)
ELSIF NOT in AND edge THEN
	edge := FALSE;
	tn := tx - tn;
	IF tn < t_short THEN
		short := TRUE;
	ELSIF tn > t_long THEN
		long := TRUE;
	ELSE
		Middle := TRUE;
	END_IF;

(* generate long pulse as soon as T_long is reached *)
ELSIF in AND tx - tn > t_long THEN
	long := TRUE;
END_IF;


(* revision history

hm	15. feb 2006	rev 1.0
	original version

hm	15 sep 2007		rev 1.1
	replaced Time() with T_PLC_MS for compatibility and performance reasons

*)
END_FUNCTION_BLOCK

(* POU Building/Jalousie/blind_night, ST *)
FUNCTION_BLOCK blind_night
VAR_INPUT
	UP, DN : BOOL;
	S_IN : BYTE;
	pi, ai : BYTE;
	E_night : BOOL := TRUE;
	E_day	: BOOL := TRUE;
	dtin : DT;
	sunrise, sunset : TOD;
END_VAR
VAR_INPUT CONSTANT
	sunrise_offset : TIME;
	sunset_offset : TIME;
	night_position : BYTE := 0;
	night_angle : BYTE := 0;
END_VAR
VAR_OUTPUT
	QU, QD : BOOL;
	status : BYTE;
	po, ao : BYTE;
END_VAR
VAR
	night : BOOL;
	last_night, last_day : DATE;
END_VAR

(*
version 1.2	6 oct 2007
programmer 	hugo
tested by		tobias


*)
IF NOT (up AND dn) AND night THEN
	(* manual operation at night will cancel operation for one night *)
	night := FALSE;
ELSIF (DT_TO_TOD(dtin) > sunset + sunset_offset) AND (last_night < DT_TO_DATE(dtin)) AND NOT night AND e_night THEN
	(* enable night *)
	night := TRUE;
	last_night := DT_TO_DATE(dtin);
ELSIF (DT_TO_TOD(dtin) > sunrise + sunrise_offset) AND (last_day < DT_TO_DATE(dtin)) AND night AND e_day AND (last_night < DT_TO_DATE(dtin)) THEN
	(* disable night *)
	night := FALSE;
	last_day := DT_TO_DATE(dtin);
END_IF;

(* shade at night only in auto mode and enable = true *)
IF UP AND DN AND night THEN
	status := 141;
	po := night_position;
	ao := night_angle;
ELSE
	QU := UP;
	QD := DN;
	po := pi;
	ao := ai;
	status := s_in;
END_IF;


(* revision history
hm	29. sep 2007	rev 1.0
	original version

hm	5. oct 2007		rev 1.1
	added enable input

hm	6. oct 2007		rev 1.2
	added pos and angle inputs and outputs
	night position and angle can now be configured
	any manual operation at night will cancel night operation

*)
END_FUNCTION_BLOCK

(* POU Time&Date/sun_time, ST *)
FUNCTION_BLOCK sun_time
VAR_INPUT
	latitude : REAL;				(* latitude of geographical position  *)
	longitude : REAL;				(* longitude of geographical position  *)
	utc : DT;						(*	world time				*)
END_VAR
VAR_OUTPUT
	sun_midday : TOD;			(*	astrological midday in hours when sun stand at south direction	*)
	sun_rise : TOD;				(*	sun rise for current day in local time *)
	sun_set : TOD;				(*	sun set for current day in local time *)
	sun_declination : REAL;		(*	sun declination at midday in degrees	*)
END_VAR
VAR
	T: INT;							(* day in the year   *)
	DK: REAL;						(* sun declination at midday *)
	delta: REAL;					(* delta from midday for sunrise and sunset  *)
	h: REAL;
	B: REAL;
	offset : REAL;
	l15: REAL;
	dat: DATE;
	last_dat: DATE;
END_VAR

(*
version 1.4	17. jan 2008
programmer 	hugo
tested by		tobias

this FUNCTION block calculates the sun rise, sun set, sun offset at midday sun declination for a given date 
for performance reasons the algorithm has been simplified and is accurate within a few minutes only 
the times are calculated in utc and have to be corrected for the given time zone
this correction is not done within sun_time because it would be a problem on days where dst is enabled or disabled


*)
dat := DT_TO_DATE(utc);
IF dat = last_dat THEN RETURN; END_IF;
last_dat := dat;
l15 := longitude * 0.0666666666666;
B := latitude * 0.0174532925199433;
h := -0.0145;
T := day_of_year(dat);
offset := -0.1752 * SIN(0.033430*T + 0.5474) - 0.1340*SIN(0.018234*T - 0.1939);
sun_midday := hour_to_tod(12 + Offset - l15);
DK := 0.40954 * SIN(0.0172 * (T-79.35));
sun_declination := deg(DK);
delta := 12*ACOS((SIN(h) - SIN(B) * SIN(DK)) / (COS(B) * COS(DK))) * 0.318309886;
sun_rise := hour_to_tod(12 - delta - Offset - l15);
sun_set := hour_to_tod(12 + delta - Offset - l15);

(* revision history

rev 1.1	hm	20.1.2007
	deleted unused variables sun_riseR and sun_setR

rev 1.2 hm 17.4.2007
	corrected error while sun:midday would not be corrected for longitude.

rev 1.3	hm	6. jan 2008
	performance improvements

rev	1.4 hm	17. jan 2008
	calculation is now only performed once a day
*)
END_FUNCTION_BLOCK

(* POU Time&Date/day_of_year, ST *)
FUNCTION day_of_year : INT
VAR_INPUT
	idate : DATE;
END_VAR
VAR
END_VAR

(*
version 1.2	4 jan 2008
programmer 	hugo
tested by		tobias

calculates the day of the year 

*)
day_of_year := DWORD_TO_INT((DATE_TO_DWORD(idate) - DATE_TO_DWORD(year_begin(year(idate))))/86400) + 1;


(* version before rev 1.2
IF step7 THEN
	day_of_year := DWORD_TO_INT(DATE_TO_DWORD(idate)/86400 + 726483 - TRUNC((year(idate)-1)*365.25));
ELSE
	day_of_year := DWORD_TO_INT(DATE_TO_DWORD(idate)/86400 + 719178 - TRUNC((year(idate)-1)*365.25));
END_IF;
*)


(* revivision history
hm	4. aug 2007		rev 1.0
	original version

hm	1. okt 2007		rev 1.1
	added compatibility to STEP7

hm	4. jan 2008		rev 1.2
	changed code for better performance
*)
END_FUNCTION

(* POU Time&Date/year_begin, ST *)
FUNCTION year_begin : DATE
VAR_INPUT
	y : INT;
END_VAR
VAR
END_VAR

(*
version 1.1	4. Jan 2008
programmer 	hugo
tested by		tobias

returs the date of january 1st for the given year  
the function works for dates from 1970 - 2099 

*)
IF Step7 THEN
	year_begin := DWORD_TO_DATE(SHR(INT_TO_DWORD(y) * 1461 - 2907389,2)*86400);
ELSE
	year_begin := DWORD_TO_DATE(SHR(INT_TO_DWORD(y) * 1461 - 2878169,2)*86400);
END_IF;

(* revision history
hm	19. dec 2007	rev 1.0
	original version

hm	4. jan 2008	rev 1.1
	formula for step7 was incorrect during leap years

*)
END_FUNCTION

(* POU Time&Date/year, ST *)
FUNCTION year : INT
VAR_INPUT
	idate : DATE;
END_VAR
VAR
END_VAR

(*
version 1.2	23 dec 2007
programmer 	hugo
tested by		tobias

returs the year of a date  
the function works for dates from 1970 - 2099 

*)
IF Step7 THEN
	year := DWORD_TO_INT((DATE_TO_DWORD(idate)+43200) / 31557600 + 1990);
ELSE
	year := DWORD_TO_INT((DATE_TO_DWORD(idate)+43200) / 31557600 + 1970);
END_IF;

(* code used prior to rev 1.1
year := DWORD_TO_INT((DATE_TO_DWORD(idate)/864+71954300)/36525);
*)

(* revision history
hm	4. aug 2006		rev 1.0
	original version

hm	1. okt 2007		rev 1.1
	corrected error in algorithm
	adjustment for S7 compatibility

hm	23.12.2007		rev 1.2
	changed code for better performance
*)
END_FUNCTION

(* POU Time&Date/hour_to_tod, ST *)
FUNCTION hour_to_tod : TOD
VAR_INPUT
	input : REAL;
END_VAR
VAR
END_VAR

(*
version 1.0	4 aug 2006
programmer 	hugo
tested by		tobias

converts an amount of hours in real to time of day 

*)
hour_to_tod := DWORD_TO_TOD(REAL_TO_DWORD(input * 3600000));
END_FUNCTION

(* POU mathematical/deg, ST *)
FUNCTION deg : REAL
VAR_INPUT
	rad : REAL;
END_VAR
VAR
END_VAR
VAR
END_VAR

(*
version 1.1	16 oct 2007
programmer 	hugo
tested by		tobias

this function converts degrees into Radiant
execution time on wago 750 - 841 =  10  us
*)
deg := modR(57.29577951308232 * Rad, 360);

(* revision history
hm	4. aug 2006		rev 1.0
	original version

hm 	16. oct 2007	rev 1.1
	added modr statement which prohibits deg to become bigger than 360

*)
END_FUNCTION

(* POU mathematical/Rad, ST *)
FUNCTION Rad : REAL
VAR_INPUT
	deg : REAL;
END_VAR
VAR
END_VAR

(*
version 1.0	4 aug 2006
programmer 	hugo
tested by	tobias

this function converts Radiant to degrees

*)
Rad := modR(0.0174532925199433 * deg,PI2);

(* revision history
hm	4. aug 2006
	original version

hm 	16. oct 2007
	added modr statement which prohibits rad to become bigger than 2PI

*)
END_FUNCTION

(* POU mathematical/modR, ST *)
FUNCTION modR : REAL
VAR_INPUT
	in : REAL;
	divi : REAL;
END_VAR

VAR
END_VAR

(*
version 1.1	4 aug 2006
programmer 	hugo
tested by		tobias

this is a modulo funtion for real numbers
modr(5.5,2.5) = 0.5


execution time on wago 750 - 841 =  29  us
*)
IF divi = 0 THEN
	modR := 0;
ELSE
	modR := in - TRUNC(in / divi) * divi;
END_IF;

(* revision history

hm 4.8.2006	rev 1.0

hm 28.1.2007	rev 1.1
	modr(x,0) will deliver the result 0

*)
END_FUNCTION

(* POU Time&Date/sun_pos, ST *)
FUNCTION_BLOCK sun_pos
VAR_INPUT
	latitude : REAL;				(* latitude of geographical position  *)
	longitude : REAL;				(* longitude of geographical position  *)
	utc : DT;						(*	world time				*)
END_VAR
VAR_OUTPUT
	B: REAL;
	HR: REAL;
END_VAR
VAR
	L: REAL;
	N: REAL; (* amount of days since 1.1.2000 12:00 *)
	G: REAL;
	K: REAL;
	A: REAL;
	X: REAL;
	D: REAL;
	TA: REAL;
	H: REAL;
	T1: REAL;
	LA: REAL;
	LO: REAL;
	SLA: REAL;
	CLA: REAL;
	CTA: REAL;
	last: DWORD;
END_VAR

(*
version 1.2	18. jan 2008
programmer 	hugo
tested by		tobias

this FUNCTION block calculates the sun position for a given date and time.
the times are calculated in utc and have to be corrected for the given time zone.
B is the angle from north and HR is the highth in degrees.

*)
(* EXIT the routine IF it was executed the 10 seconds which is equal to 0.04 degrees accuracy *)
IF T_PLC_MS() - last < 10000 THEN RETURN; END_IF;
last := T_PLC_MS();

(* calculate the angles *)
N := (DT_TO_DWORD(utc) - 946728000)/86400;
LA := Rad(latitude);
SLA := SIN(LA);
CLA := COS(LA);
LO := Rad(longitude);
L := modR(280.460 + 0.9856474 * N,360);
G := Rad(modR(357.528 + 0.9856003 * N,360));
K := Rad(L + 1.915 * SIN(G) + 0.02 * SIN(2*G));
X := Rad(23.439 - 0.0000004 * N);
A := ATAN(COS(X)*TAN(K));
IF COS(K) < 0 THEN A := A + PI1; END_IF;
D := ASIN(SIN(X) * SIN(K));
TA := Rad(modR(6.697376 + 0.065709825 * (TRUNC(N - 0.5) + 0.5) + TOD_TO_REAL(DT_TO_TOD(utc)) * 2.78538333E-7, 24) * 15 + longitude - deg(A));
CTA := COS(TA);
T1 := CTA*SLA - TAN(D)*CLA;
B := deg(ATAN(SIN(TA)/T1));
IF T1 < 0 THEN B := B + 180; END_IF;
IF B > 180 THEN
	B := B - 180;
ELSIF B < 180 THEN
	B := B + 180;
END_IF;
H := deg(ASIN(COS(D)*CTA*CLA+SIN(D)*SLA));
HR := H + 0.017 / TAN(Rad(H+10.3/(H+5.11)));


(* revision history
hm	1. feb 2007	rev 1.0
	original version

hm	6. jan 2008	rev 1.1
	performance improvements

hm	18. jan 2008	rev 1.2
	further performance improvements
	only calculate once every 10 seconds
*)
END_FUNCTION_BLOCK

(* POU Building/Jalousie/BLIND_SHADE, ST *)
FUNCTION_BLOCK BLIND_SHADE
VAR_INPUT
	UP, DN : BOOL;
	S_IN : BYTE;
	pi, ai : BYTE;
	enable : BOOL;
	sun : BOOL;
	dtin : DT;
	sunrise, sunset : TOD;
	sun_hor, sun_ver : REAL;
END_VAR
VAR_INPUT CONSTANT
	sunrise_offset : TIME := T#1h;
	sunset_preset : TIME := T#1h;
	direction : REAL := 180;
	angle_offset : REAL := 80;
	slat_width : REAL := 80;
	Slat_spacing : REAL := 60;
	Shade_delay : TIME := T#60s;
END_VAR
VAR_OUTPUT
	QU, QD : BOOL;
	status : BYTE;
	po, ao : BYTE;
END_VAR
VAR
	angle: REAL;
	sun_delay : TOF;
END_VAR

(*
version 1.2	24 nov 2007
programmer 	hugo
tested by		tobias


*)
(* the input sun is sent through tof which will delay the shade for the time shade_delay *)
sun_delay(IN := sun, PT := shade_delay);

IF UP AND DN AND enable AND sun_delay.Q AND sun_hor > direction - angle_offset AND sun_hor < direction + angle_offset AND
	DT_TO_TOD(dtin) > sunrise + sunrise_offset AND DT_TO_TOD(dtin) < sunset - sunset_preset THEN
	status := 151;
	QU := UP;
	QD := DN;
	(* position is fully down *)
	po := 0;
	(* shading is active now calculate the slat angle *)
	(* calculate the max angle for the blind *)
	angle := deg(ATAN(slat_spacing / slat_width));
	(* check if sun angle is between 0 and max angle *)
	IF sun_ver > 0 AND sun_ver < angle THEN
		angle := sun_ver + deg(ACOS(COS(Rad(sun_ver))*slat_spacing / Slat_width));
		ao := INT_TO_BYTE(LIMIT(0,TRUNC(angle * 255 / 90), 255));
	ELSE
		ao := 255;
	END_IF;
ELSE
	QU := UP;
	QD := DN;
	po := pi;
	ao := ai;
	status := S_IN;
END_IF;

(* revision history
hm	15 oct. 2007	rev 1.0
	original version

hm	19. oct 2007	rev 1.1
	manual mode was not detected because outputs were checked and not inputs UP and DN

hm	24. nov 2007	rev 1.2
	added shade_delay to avoid constant up and down if sun is out parcially
*)
END_FUNCTION_BLOCK

(* POU XTEST/Baustein Tests/control_test, CFC *)
PROGRAM control_test
VAR
	Offset : REAL;
	x1: FT_PT1;
	step: REAL;
	t1: TIME := T#1s;
	Out: REAL;
	x2: FT_PT2;
	d: REAL := 0.5;
	out2: REAL;
	x3: FT_PID;
	TV, TN : REAL := 1;
	out3: REAL;
	SET: REAL;
	x4: FT_PI;
	M_in: REAL;
	M_en: BOOL;
	RST: BOOL;
	INTB: REAL := 10;
	KP: REAL := 1;
	KI: REAL := 1;
	L_L: REAL := -1000;
	L_H: REAL := 1000;
	out4: REAL;
	l1: BOOL;
	o1: BOOL;
	l2: BOOL;
	o2: BOOL;
	x5: FT_PT1;
END_VAR
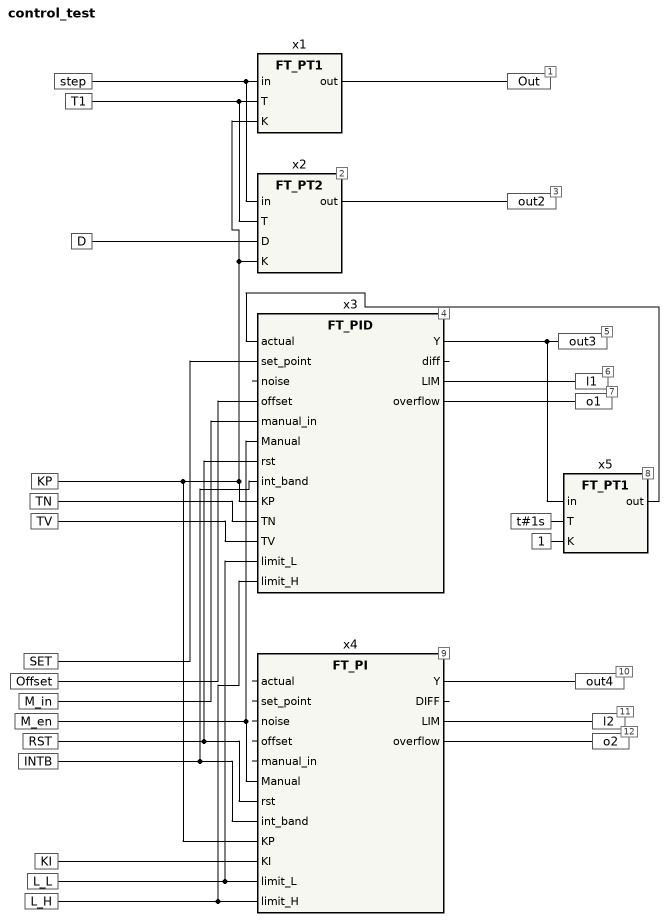
_CFC_ (* Continuous Function Chart, elements in execution order *)
#0 x1:FT_PT1(in: step, T: T1, K: KP)
#1 Out <= #0.out
#2 x2:FT_PT2(in: step, T: T1, D: D, K: KP)
#3 out2 <= #2.out
#4 x3:FT_PID(actual: #8.out, set_point: SET, noise: -, offset: Offset, manual_in: M_in, Manual: M_en, rst: RST, int_band: INTB, KP: KP, TN: TN, TV: TV, limit_L: L_L, limit_H: L_H)
#5 out3 <= #4.Y
#6 l1 <= #4.LIM
#7 o1 <= #4.overflow
#8 x5:FT_PT1(in: #4.Y, T: t#1s, K: 1)
#9 x4:FT_PI(actual: -, set_point: -, noise: -, offset: -, manual_in: -, Manual: M_en, rst: RST, int_band: INTB, KP: KP, KI: KI, limit_L: L_L, limit_H: L_H)
#10 out4 <= #9.Y
#11 l2 <= #9.LIM
#12 o2 <= #9.overflow
_END_CFC_
(* the same logic as Structured Text *)
x1(in := step, T := T1, K := KP);
Out := x1.out;
x2(in := step, T := T1, D := D, K := KP);
out2 := x2.out;
x3(actual := x5.out, set_point := SET, offset := Offset, manual_in := M_in, Manual := M_en, rst := RST, int_band := INTB, KP := KP, TN := TN, TV := TV, limit_L := L_L, limit_H := L_H);
out3 := x3.Y;
l1 := x3.LIM;
o1 := x3.overflow;
x5(in := x3.Y, T := t#1s, K := 1);
x4(Manual := M_en, rst := RST, int_band := INTB, KP := KP, KI := KI, limit_L := L_L, limit_H := L_H);
out4 := x4.Y;
l2 := x4.LIM;
o2 := x4.overflow;
END_PROGRAM

(* POU engineering/control/FT_PT1, ST *)
FUNCTION_BLOCK FT_PT1
VAR_INPUT
	in : REAL;
	T : TIME;
	K : REAL := 1;
END_VAR
VAR_OUTPUT
	out : REAL;
END_VAR
VAR
	last : DWORD;
	tx: DWORD;
	init: BOOL;
END_VAR

(*
version 1.7	5 jan 2008
programmer 	hugo
tested by		tobias

FT_PT1 is an low pass filter with a programmable time T and faktor K.
 
*)
(* read system time *)
tx := T_PLC_US();

(* startup initialisation *)
IF NOT init THEN
	last := tx;
	init := TRUE;
	out := K * in;
ELSIF T = t#0s THEN
	out := K * in;
ELSE
	out := out + (in * K - out) * (Tx - last) / TIME_TO_REAL(T) * 1E-3;
END_IF;
last := tx;

(*
hm 1.1.2007	rev 1.1
	corrected error while startup value was not correct
	for very small time values real output would run out of range.

hm 3.1.2007	rev 1.2
	corrected an error for falling edge failures.
	added output faktor K.

hm 27. 2. 2007	rev 1.3
	output will be input during init for definitive startup condition.

hm	15.9.2007	rev 1.4
	changed time() to T_PLC_US() for compatibilitxy resons
	increased internal accuracy to Microseconds instead of Milliseconds

hm	23. oct 2007	rev 1.5
	added out := in to the init statements

hm	30. nov 2007	rev 1.6
	changed out to be K * in during initialization

hm	5. jan 2008		rev 1.7
	improved code for better performance
*)
END_FUNCTION_BLOCK

(* POU engineering/measurements/T_PLC_US, ST *)
FUNCTION T_PLC_US : DWORD
VAR CONSTANT
	debug : BOOL := FALSE;
	N : INT := 0;
	offset : DWORD := 0;
END_VAR
VAR
	tx : TIME;
	temp : DWORD := 1;
END_VAR

(*
version 1.1	12 nov 2007
programmer 	hugo
tested by		tobias

T_PLC_US reads the internal PLC timer and return the time, it has the advantage to be able to set a debug mode 
and speed up the counter to test the plc timer overrun which occurs every 50 days respectively 25 days at siemens S7
this routine also allows to correct the behavior of s7 where the internal plc counter will not count all 32 bits.

*)
tx := TIME();
T_PLC_US := TIME_TO_DWORD(Tx)*1000;
(* hier muss die korrektur für step7 stattfinden
plctime muss den vollen wertebereich von time ausnutzen:
wenn bei step7 time -24tage bis plus 24 tage ist dann muss der timer auch beim überlauf auf -24tage springen 
und auf keinen fall auf 0 !!!!
für siemens muss ein weiterer fb im main eingebunden werden der sicherstellt das alle 32 bits durchgezählt werden.
es kann nur ein fb sein den er muss sich das oberste (32te) bit merken.
oder etwa spring s7 bei überlauf auf -24 tage????? dann wäre keine korrektur nötig.
*)
IF debug THEN
	T_PLC_US := (SHL(T_PLC_US,N) OR SHL(temp,N)-1) + Offset;
END_IF;

(* revision history
hm	14.9.2007	rev 1.0
	original version

hm	12. nov 2007	rev 1.1
	added temporaray variable tx because some compilers could not handle time() as an argument

*)
END_FUNCTION

(* POU engineering/control/FT_PT2, ST *)
FUNCTION_BLOCK FT_PT2
VAR_INPUT
	in : REAL;
	T : TIME;
	D : REAL;
	K : REAL := 1;
END_VAR
VAR_OUTPUT
	out : REAL;
END_VAR
VAR
	init: BOOL;
	int1 : FT_INT;
	int2 : FT_INT;
	tn: REAL;
END_VAR

(*
version 1.3	30 Nov 2007
programmer 	hugo
tested by		tobias

FT_PT2 is a 2nd grade filter with programmable times T, D and faktor K.
 
*)
(* startup initialisation *)
IF NOT init THEN
	out := K * in;
	init := TRUE;
ELSIF T = t#0s THEN
	out := K * in;
ELSE
	tn := TIME_TO_REAL(T)/1000;
	int1(in := in * K / (TN * TN) - int1.Out * 2 *D / TN - int2.Out / (TN * TN));
	int2(in := int1.Out);
	out := int2.out;
END_IF;

(* revision history

15.1.2007 hm		rev 1.1
	changed formula to new more acurate formula
	old code:
	tx := TIME();
	IF NOT init THEN
		last := tx;
		init := TRUE;
	ELSE
		IF T> t#0s THEN
			out1 := out1 + (in - out1) * TIME_TO_REAL(Tx - last) / TIME_TO_REAL(T);
		ELSE
			out1 := in;
		END_IF;
		IF T > t#0s THEN
			out2 := out2 + (out1 - out2) * TIME_TO_REAL(Tx - last) / TIME_TO_REAL(T);
		ELSE
			out2 := out1;
		END_IF;
		out := out2 * K;
	END_IF;
	last := tx;

hm 		15.9.2007		rev 1.2
	deleted unused code for init system time reading tx	

hm		30.11.2007		rev 1.3
	changed out to be K * in during initialization
	avoind divide by 0 if tn = 0
*)
END_FUNCTION_BLOCK

(* POU engineering/control/FT_INT, ST *)
FUNCTION_BLOCK FT_INT
VAR_INPUT
	in : REAL;
	K : REAL := 1;
	run : BOOL := 1;
	rst: BOOL := 0;
	out_min : REAL := -1E-37;
	out_max : REAL := 1E37;
END_VAR
VAR_OUTPUT
	Out : REAL;
END_VAR
VAR
	last: DWORD;
	in_last : REAL;
	tx: DWORD;
	init: BOOL;
	tc: DWORD;
	out1: REAL;
	out2: REAL;
	tmp: REAL;
END_VAR


(*
version 1.7	8. feb 2008
programmer 	hugo
tested by		tobias

FT_int is an integrator with input IN and factor K.
integration is only done while run = true, if run is false integration is stopped and the out remains at the last value.
if run is left unconnected, run is considered true by the function block.
the output ET will display the total integration time from last reset.
a rst input will reset output and the timer ET to 0.
the out_min and out_max values can be set to ,imit the output value range. 
the default for K is 1.

 
*)
(* read and store system time *)
tx := T_PLC_US();
tc := tx - last;

(* startup initialisation *)
IF rst OR NOT init THEN
	out1 := 0;
	out2 := 0;
	init := TRUE;
	last := tx;
ELSIF run AND tc > 0 THEN
	last := tx;
	out1 := out1 + (in + in_last) * tc * K * 5E-7;
	tmp := in * K * 10000;
	IF out1 > tmp THEN
		out1 := out1 - tmp;
		out2 := out2 + tmp;
	END_IF;
ELSIF NOT run THEN
	last := tx;
END_IF;
in_last := in;
out := LIMIT(out_min, out1 + out2, out_max);

(*
hm 13.12.2006	rev 1.1
	changed to "trapezregel" which increases accuracy
	before out := out + in * time new: out := out + (in + in_last) / 2 * time

hm 15.1.2007		rev 1.2
	added default for k to be 1.

hm	15.9.2007		rev 1.3
	replaced time() with T_PLC_US for compatibility and performance reason
	increased internal accuracy to microseconds

hm 29. oct 2007		rev 1.4
	changed code so int will not be called is time difference is 0 to increase accuracy on systems
	with cycle times below 1ms

hm	2. dec 2007	 	rev 1.5
	changed code for better performance

hm	5. jan 2008		rev 1.6
	further improvements in performance

hm	8. feb 2008		rev 1.7
	deleted limits +/- 1000 now limit is the range of real
	added variables out1 and out2 to extend the resolution
	corrected an error with elapsed time
	deleted unusfull output ET
*)
END_FUNCTION_BLOCK

(* POU engineering/control/FT_PID, ST *)
FUNCTION_BLOCK FT_PID
VAR_INPUT
	actual, set_point, noise, offset, manual_in : REAL;
	Manual : BOOL;
	rst : BOOL := FALSE;
	int_band : REAL := 100;
	KP : REAL := 1.0;
	TN : REAL := 1.0;
	TV : REAL := 1.0;
	limit_L : REAL := -1000;
	limit_H : REAL := 1000;
END_VAR
VAR_INPUT CONSTANT
	int_limit_L : REAL := -1000;
	int_limit_H : REAL := 1000;
END_VAR
VAR_OUTPUT
	Y : REAL;
	diff: REAL;
	LIM, overflow : BOOL;
END_VAR
VAR
	integ : FT_INT;
	deriv : FT_deriv;
END_VAR

(*
version 1.6	5 jan 2008
programmer 	hugo
tested by		tobias

FT_PID is a pid controller with manual functionality.
The PID controller works according to the fomula Y = KP * ( e + 1/TN * INTEG(e) + TV *DERIV(e)) + offset, while e = set_point - actual.
a rst will reset all internal data, while a switch to manual will cause the controller to follow the function Y = manual_in + offset.
limit_h and Limit_l set the possible output range of Y.
the output flags lim will signal that the output limits are active and overflow will signal that the integrator has reached the max or min limit.  

since rev 1.1 the "trapezregel is used for more accuracy.
rev 1.2 added selective integratin which means the integrative component is only active within a small range of the target value 
this avoids the integrator to go to limits while an input setpoint change happened and is only causing overshoots.
the int_band is by default 100 which means the int is active all the time and if set to for example to 0.1 the integrator is only active
while the input is between 0.9 and 1.1 of the set_point value.

default values for KP = 1, TN = 1, TV = 1, LIMIT_L = -1000, LIMIT_H = +1000.
*)
IF NOT rst AND NOT manual THEN
	(* calculate the process error *)
	DIFF := dead_band(set_point - actual, Noise);
	IF ABS(diff) <= int_band AND NOT overflow AND TN > 0 THEN
		(* integrator is within int_band and needs to be run *)
		integ(in := diff, K := 1/TN, run := TRUE, rst := FALSE, out_min := int_limit_L, out_max := int_limit_H);
		(* check if integrator has reached its limits and set overflow *)
		IF integ.Out >= int_limit_H OR integ.Out <= int_limit_L THEN overflow := TRUE; END_IF;
	ELSE
		(* int_band is exceeded, integrator needs to be cleared *)
		integ(rst := TRUE);
	END_IF;
	(* calculate the derivative part *)
	deriv(in := diff, K := TV);
	(* add up all parts *)
	Y := KP * (integ.Out + deriv.out + diff);
ELSIF rst THEN
	integ(rst := TRUE);		(* reset the integrator *)
	overflow := FALSE;		(* clear the overflow flag *)
	Y := (limit_H + Limit_L) * 0.5 - Offset;	(* set the output between limit_L and limit_L offset will be added again at the end *)
ELSIF manual THEN
	Y := manual_in;
	integ(rst := TRUE);		(* make sure integrator is reset to 0 *)
	overflow := FALSE;		(* manual operation will cancel overflow because integrator was reset *)
END_IF;

(* add offset to Y *)
Y := Y + Offset;

(* limit the outputs and set the lim flag if necessary *)
IF y > limit_H THEN
	y := limit_H;
	lim := TRUE;
ELSIF y < limit_L THEN
	y := limit_L;
	lim := TRUE;
ELSE
	lim := FALSE;
END_IF;


(* old code before rev 1.4
IF rst OR KP = 0 THEN
	y := Offset;
	integ(rst := 1);
	integ.rst := 0;
ELSIF manual THEN
	Y := manual_in + Offset;
	integ(rst := 1);
	integ.rst := 0;
ELSE
	(* calcualtion of the actual PID values *)
	diff := set_point - actual;

	(* integrator is only called if TN > 0 and input is within int_band othewrwise it is disabled *)
	IF TN > 0 AND actual > set_point - int_band AND actual < set_point + int_band THEN
		integ(in := diff, K := 1/TN, out_min := (limit_L - offset) / KP, out_max := (limit_H - offset) / KP);
	ELSE
		integ(rst := 1);
		integ.rst := 0;
	END_IF;
	deriv(in := diff, K := TV);

	(* check if integrator has reached the allowed limits and set overflow if necessary *)
	IF integ.Out >= (limit_H - offset) / KP THEN
		Y := limit_H;
		overflow := TRUE;
	ELSIF integ.Out <= (limit_L - offset) / KP THEN
		Y := limit_L;
		overflow := TRUE;
	ELSE
		Y := KP * (integ.Out + deriv.out + diff) + offset;
		overflow := FALSE;
	END_IF;

	(* this portion limits the output to limit_H and limit_L and set the lim flag if limits are exceeded *)
	IF Y > limit_H THEN
		Y := limit_H;
		Lim := TRUE;
	ELSIF Y < limit_L THEN
		Y := limit_L;
		lim := TRUE;
	ELSE
		lim := FALSE;
	END_IF;
END_IF;
*)

(* revision history

hm 1.12.2006	 	rev 1.1
	changed algorithm to trapezregel for higher accuracy.

hm 3.1.2007		rev 1.2
	added integ_band to select when the integrator is active.

hm	3.3.2007		rev 1.3
	added default values to inputs KP, TN, TV, LIMIT_L und LIMIT_H.

hm 31.oct 2007	rev 1.4
	total rewrite of the module to avoid failures when one of the limits is 0

hm	3.11.2007	rev 1.5
	added noise input to filter noise
	added output diff
	set limit output false when output is within limits
	overfolw was not set correctly

hm	5. jan 2008	rev 1.6
	improved code for better performance
*)
END_FUNCTION_BLOCK

(* POU engineering/control/FT_deriv, ST *)
FUNCTION_BLOCK FT_deriv
VAR_INPUT
	in : REAL;
	K : REAL := 1;
	run : BOOL := 1;
END_VAR
VAR_OUTPUT
	out : REAL;
END_VAR
VAR
	old: REAL;
	tx: DWORD;
	last: DWORD;
	init: BOOL;
END_VAR


(*
version 1.3	29 oct 2007
programmer 	hugo
tested by		tobias

FT_deriv calculates the derivate over the signal "in" with Faktor "K".
a run input enables or stops the calculation, if left unconnected its true and therfore the calculation is executed.
if K is not specified the default is 1.

*)
(* read system time *)
tx := T_PLC_US();

(* init on firsat startup *)
IF NOT init THEN
	init := TRUE;
	old := in;
	last := tx;
END_IF;
IF run AND tx - last > 0 THEN
	out := (in - old) / DWORD_TO_REAL(tx - last) * 1000000.0 * K;
	last := tx;
ELSE
	out := 0;
	last := tx;
END_IF;
old := in;


(*
hm 3.1.2007			rev 1.1
	added init code for startup
	set the default for K to 1

hm	15. sep 2007	rev 1.2
	replaced Time() with T_PLC_US for compatibility and performance reasons
	increased accuracy and work in microseconds internally

hm 29 oct 2007	rev 1.3
	prohibit calculation when tx - last = 0 to avoid division by 0 and increase accuracy on fast systems
*)
END_FUNCTION_BLOCK

(* POU engineering/control/dead_band, ST *)
FUNCTION dead_band : REAL
VAR_INPUT
	X : REAL;
	L : REAL;
END_VAR
VAR
END_VAR

(*
version 1.0	2 nov 2007
programmer 	hugo
tested by		tobias

DEAD_BAND ist eine lineare Übertragungsfunktion mit Totzone. Die Funktion verschiebt den positiven Teil der Kurve um +L und den negativen Teil der Kurve um -L.
DEAD_BAND = X wenn Abs(X) > L wenn Abs(X) > L
DEAD_BAND = 0 wenn Abs(X) <= L

*)
IF ABS(x) > L THEN
	dead_band := X - sgn(x) * L;
ELSE
	dead_band := 0;
END_IF;

(* revision history
hm		2.11.07	rev 1.0
	original version
*)
END_FUNCTION

(* POU mathematical/sgn, ST *)
FUNCTION sgn : INT
VAR_INPUT
	X : REAL;
END_VAR
VAR
END_VAR

(*
version 1.1	11 nov 2007
programmer 	hugo
tested by	tobias

sgn returns 0 when X = 0 , -1 when X < 1 and +1 when X > 1

*)
IF X > 0 THEN
	sgn := 1;
ELSIF X < 0 THEN
	sgn := -1;
ELSE
	sgn := 0;
END_IF;

(* revision histroy
hm	16. oct 2007	rev 1.0
	original version

hm	11. nov 2007	rev 1.1
	changed type of function from real to int
*)
END_FUNCTION

(* POU engineering/control/FT_PI, ST *)
FUNCTION_BLOCK FT_PI
VAR_INPUT
	actual, set_point, noise, offset, manual_in : REAL;
	Manual : BOOL;
	rst : BOOL := FALSE;
	int_band : REAL := 100;
	KP : REAL := 1.0;
	KI : REAL := 1.0;
	limit_L : REAL := -1000;
	limit_H : REAL := 1000;
END_VAR
VAR_INPUT CONSTANT
	int_limit_L : REAL := -1000;
	int_limit_H : REAL := 1000;
END_VAR
VAR_OUTPUT
	Y : REAL;
	DIFF : REAL;
	LIM, overflow : BOOL;
END_VAR
VAR
	integ : FT_INT;
END_VAR

(*
version 1.2	5 jan 2008
programmer 	hugo
tested by		tobias

FT_PI is a PI controller with manual functionality.
The PID controller works according to the fomula Y = e *(KP+ KI * INTEG(e) ) + offset, while e = set_point - actual.
a rst will reset all internal data, while a switch to manual will cause the controller to follow the function Y = manual_in + offset.
limit_h and Limit_l set the possible output range of Y.
the output flags lim will signal that the output limits are active and overflow will signal that the integrator has reached its limits.

since rev 1.1 the "trapezregel is used for more accuracy.
rev 1.2 added selective integratin which means the integrative component is only active within a small range of the target value 
this avoids the integrator to go to limits while an input setpoint change happened and is only causing overshoots.
the int_band is by default 100 which means the int is active all the time and if set to for example to 0.1 the integrator is only active
while the input is between 0.9 and 1.1 of the set_point value.

default values for KP = 1, TN = 1, TV = 1, LIMIT_L = -1000, LIMIT_H = +1000.
*)
IF NOT rst AND NOT manual THEN
	(* calculate the process error *)
	DIFF := dead_band(set_point - actual, Noise);
	IF ABS(diff) <= int_band AND NOT overflow THEN
		(* integrator is within int_band and needs to be run *)
		integ(in := diff, K := KI, run := TRUE, rst := FALSE, out_min := int_limit_L, out_max := int_limit_H);
		(* check if integrator has reached its limits and set overflow *)
		IF integ.Out >= int_limit_H OR integ.Out <= int_limit_L THEN overflow := TRUE; END_IF;
	ELSE
		(* int_band is exceeded, integrator needs to be cleared *)
		integ(rst := TRUE);
	END_IF;
	Y := KP * diff + integ.Out;
ELSIF rst THEN
	integ(rst := TRUE);		(* reset the integrator *)
	overflow := FALSE;		(* clear the overflow flag *)
	Y := (limit_H + Limit_L) * 0.5 - Offset;	(* set the output between limit_L and limit_L offset will be added again at the end *)
ELSIF manual THEN
	Y := manual_in;
	integ(rst := TRUE);		(* make sure integrator is reset to 0 *)
	overflow := FALSE;		(* manual operation will cancel overflow because integrator was reset *)
END_IF;

(* add offset to Y *)
Y := Y + Offset;

(* limit the outputs and set the lim flag if necessary *)
IF y > limit_H THEN
	y := limit_H;
	lim := TRUE;
ELSIF y < limit_L THEN
	y := limit_L;
	lim := TRUE;
ELSE
	lim := FALSE;
END_IF;



(* revision history
hm 	31.10.2007 	rev 1.0
	original version

hm	3.11.2007	rev 1.1
	added noise input to filter noise
	added output diff
	set limit output false when output is within limits
	overfolw was not set correctly

hm	5. jan 2008	rev 1.2
	improved performance
*)
END_FUNCTION_BLOCK

(* POU XTEST/Baustein Tests/crc_test, CFC *)
PROGRAM crc_test
VAR
	arr : ARRAY[1..9] OF BYTE := 49, 50, 51, 52, 53, 54, 55, 56, 57;
	code: DWORD;
	hex: STRING;
END_VAR
VAR (* helpers for the ST form of the networks *)
	_t1 : DWORD;
END_VAR
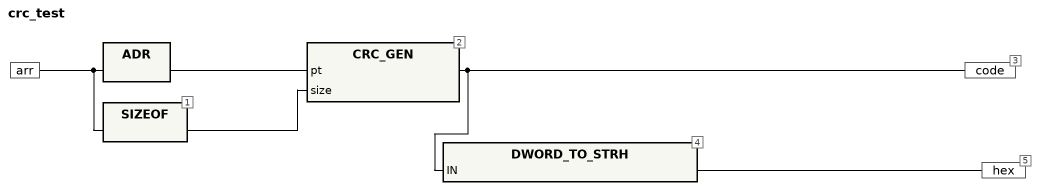
_CFC_ (* Continuous Function Chart, elements in execution order *)
#0 ADR(arr)
#1 SIZEOF(arr)
#2 CRC_GEN(pt: #0, size: #1, Polynom_L := 263, init := 255, XOR_out := 255, rev_in := TRUE, rev_out := TRUE)
#3 code <= #2
#4 DWORD_TO_STRH(IN: #2)
#5 hex <= #4
_END_CFC_
(* the same logic as Structured Text *)
_t1 := CRC_GEN(ADR(arr), SIZEOF(arr));
code := _t1;
hex := DWORD_TO_STRH(IN := _t1);
END_PROGRAM

(* POU Logic/Others/CRC_GEN, ST *)
FUNCTION CRC_GEN : DWORD

VAR_INPUT
	pt : POINTER TO ARRAY[0..32000] OF BYTE;
	size : INT;
END_VAR
VAR_INPUT CONSTANT
	Polynom_L : DWORD;
	Polynom_32 : BOOL;
	init: DWORD := 0;
	XOR_out : DWORD;
	rev_in : BOOL;
	rev_out : BOOL;
END_VAR
VAR
	polynom : DWORD;
	p_length : INT;
	BS : BYTE;
	data : DWORD;
	count : BYTE;
	temp : BOOL;
	step: INT;
	s4: INT;
END_VAR

(*
version 1.3	2 jan 2008
programmer 	hugo
tested by		tobias

CRC_GEN generates a CRC checksum from a block of data and returns  the checksum in a DWORD to be connected to the data for transmission.
the CRC Polynom is specified with the config variable Polynom_L which holds the lowest 32 bits of the polynom and Polynom_33 which holds bit 33 of the Polynom.
A Polynom x4 + X + 1 is represented by 10011.
The input data is an array of byte of any size, the function is called by CRC_GEN(ADR(array),SIZEOF(array)).

*)
(* check for polynom length and calculate p_length polynom will be aligned to high side of word*)
polynom := polynom_L;
IF polynom_32 THEN
	p_length := 33;
ELSE;
	p_length := 32;
	WHILE p_length > 0 AND NOT polynom.31 DO
		p_length := p_length - 1;
		Polynom := SHL(polynom,1);
	END_WHILE;
	Polynom := SHL(polynom,1);
END_IF;


(* load start code and first data byte for crc calculation *)
data := init;
IF rev_in THEN bs := reverse(pt^[0]); ELSE bs := pt^[0]; END_IF;

(* calcualte checksum *)
s4 := size + 4;
WHILE step < s4 DO
	temp := data.31;
	data := SHL(data,1);
	data.0 := BS.7;
	bs := SHL(bs,1);
	count := count + 1;
	IF count = 8 THEN
		step := step + 1;
		count := 0;
		IF step < size THEN
			IF rev_in THEN bs := reverse(pt^[step]); ELSE bs := pt^[step]; END_IF;
		END_IF;
	END_IF;
	(* check highest bit if true then xor polynom *)
	IF temp THEN data := data XOR polynom; END_IF;
END_WHILE;

(* reverse crc if necessary *)
IF rev_out THEN
	CRC_GEN.31 := data.31;
	FOR step := p_length TO 3 BY -1 DO
		data := SHL(data,1);
		CRC_GEN := SHR(CRC_GEN,1);
		CRC_GEN.31 := data.31;
	END_FOR;
ELSE
	CRC_GEN := data;
END_IF;

(* final XOR and align crc checksum to right side of dword *)
CRC_GEN := CRC_GEN XOR SHL(xor_out, 33 - p_length);
CRC_GEN := SHR(CRC_GEN,33 - p_length);


(* old code prior to rev 1.2
B1 := pt^[0];
IF size > 1 THEN B2 := pt^[1]; ELSE B2 := 0; END_IF;
IF size > 2 THEN B3 := pt^[2]; ELSE B3 := 0; END_IF;
IF size > 3 THEN B4 := pt^[3]; ELSE B4 := 0; END_IF;
IF size > 4 THEN BS := pt^[4]; ELSE BS := 0; END_IF;
data := DWord_of_Byte(B4,B3,B2,B1);

WHILE step < size DO
	temp := data.31;
	data := SHL(data,1);
	data.0 := BS.7;
	bs := SHL(bs,1);
	count := count + 1;
	IF count = 8 THEN
		step := step + 1;
		count := 0;
		IF step + 4 < size THEN bs := pt^[step+ 4]; END_IF;
	END_IF;
	(* check highest bit if true then xor polynom *)
	IF temp = TRUE THEN
		data := data XOR polynom;
	END_IF;
END_WHILE;

(* align crc checksum to right side of dword *)
CRC_GEN := SHR(data,32 - p_length +1);
*)


(* typical crc polynoms

CRC-4-ITU 			x4 + x + 1 					(ITU G.704, p. 12) 	0x3 or 0xC (0x9)
CRC-5-ITU 			x5 + x4 + x2 + 1 			(ITU G.704, p. 9) 	0x15 or 0x15 (0x0B) Bluetooth
CRC-5-USB 			x5 + x2 + 1 				(use: USB token packets) 	0x05 or 0x14 (0x9)
CRC-6-ITU 			x6 + x + 1 					(ITU G.704, p. 3) 	0x03 or 0x30 (0x21)
CRC-7 				x7 + x3 + 1 				(use: telecom systems, MMC) 	0x09 or 0x48 (0x11)
CRC-8-ATM 			x8 + x2 + x + 1 				(use: ATM HEC) 	0x07 or 0xE0 (0xC1)
CRC-8-CCITT 		x8 + x7 + x3 + x2 + 1 		(use: 1-Wire bus) 	0x8D or 0xB1 (0x63)
CRC-8-Dallas/Maxim 	x8 + x5 + x4 + 1 			(use: 1-Wire bus) 	0x31 or 0x8C (0x19)
CRC-8 				x8 + x7 + x6 + x4 + x2 + 1 	0xD5 or 0xAB (0x57)
CRC-8-SAE J1850 	x8 + x4 + x3 + x2 + 1 		0x1D or 0xB8
CRC-10 				x10 + x9 + x5 + x4 + x + 1 	0x233 or 0x331 (0x263)
CRC-12 				x12 + x11 + x3 + x2 + x + 1 (use: telecom systems) 	0x80F or 0xF01 (0xE03)
CRC-15-CAN 			x15 + x14 + x10 + x8 + x7 + x4 + x3 + 1 	0x4599 or 0x4CD1 (0x19A3)
CRC-16-Fletcher 	Not a CRC; see Fletcher's checksum 	Used in Adler-32 A & B CRCs
CRC-16-CCITT 	x16 + x12 + x5 + 1 (XMODEM,X.25, V.41, Bluetooth, PPP, IrDA; known as "CRC-CCITT") 	0x1021 or 0x8408 (0x0811)
CRC-16-IBM 	x16 + x15 + x2 + 1 (USB, many others; also known as "CRC-16") 	0x8005 or 0xA001 (0x4003)
CRC-24-Radix-64 	x24 + x23 + x18 + x17 + x14 + x11 + x10 + x7 + x6 + x5 + x4 + x3 + x + 1 	0x864CFB or 0xDF3261 (0xBE64C3)
CRC-32-Adler 	Not a CRC; see Adler-32 	See Adler-32
CRC-32-MPEG2 	x32 + x26 + x23 + x22 + x16 + x12 + x11 + x10 + x8 + x7 + x5 + x4 + x2 + x + 1 	0x04C11DB7 or 0xEDB88320 (0xDB710641) Also used in IEEE 802.3
CRC-32-IEEE 802.3 	x32 + x26 + x23 + x22 + x16 + x12 + x11 + x10 + x8 + x7 + x5 + x4 + x2 + x + 1 (V.42) 	0x04C11DB7 or 0xEDB88320 (0xDB710641)
CRC-32C (Castagnoli) 	x32 + x28 + x27 + x26 + x25 + x23 + x22 + x20 + x19 + x18 + x14 + x13 + x11 + x10 + x9 + x8 + x6 + 1 	0x1EDC6F41 or 0x82F63B78 (0x05EC76F1)
CRC-64-ISO 	x64 + x4 + x3 + x + 1 (use: ISO 3309) 	0x000000000000001B or 0xD800000000000000 (0xB000000000000001)
CRC-64-ECMA-182 	x64 + x62 + x57 + x55 + x54 + x53 + x52 + x47 + x46 + x45 + x40 + x39 + x38 + x37 + x35 + x33 + x32 + x31 + x29 + x27 + x24 + x23 + x22 + x21 + x19 + x17 + x13 + x12 + x10 + x9 + x7 + x4 + x + 1
(as described in ECMA-182 p.63) 	0x42F0E1EBA9EA3693 or 0xC96C5795D7870F42 (0x92D8AF2BAF0E1E85)

*)

(* revision history

hm		9.6.2007	rev 1.0		
	original version 

hm		11.9.2007	rev 1.1
	deleted unused variable i

hm		9. oct 2007 rev 1.2
	added init code for crc and xor_out
	added refelct in and reflect_out (rev_in und Rev_out)

hm		2. jan 2008	rev 1.3
	small changes for performance improvements
*)
END_FUNCTION

(* POU Logic/gate logic/reverse, ST *)
FUNCTION reverse : BYTE
VAR_INPUT
	IN : BYTE;
END_VAR
VAR
END_VAR

(*
	version 1.0	9. oct 2006
	programmer 	hugo
	tested BY		tobias

This function reverses the bits of a byte so that after execution bit 7 is at bit 0 location and so forth.

*)
reverse.7 := in.0;
reverse.6 := in.1;
reverse.5 := in.2;
reverse.4 := in.3;
reverse.3 := in.4;
reverse.2 := in.5;
reverse.1 := in.6;
reverse.0 := in.7;


(* revision history
hm		9.oct 2007	rev 1.0
	original version

*)
END_FUNCTION

(* POU String/DWORD_TO_STRH, ST *)
FUNCTION DWORD_TO_STRH : STRING
VAR_INPUT
	IN : DWORD;
END_VAR
VAR
	i : INT;
	temp : BYTE;
	pt : POINTER TO BYTE;
END_VAR

(*
version 1.2	15 dec 2007
programmer 	hugo
tested by		tobias

DWORD_TO_STRINGH converts a DWORD to a String of Hexadecimal represented by '0' .. '9' and 'A' .. 'F'.
The lowest order Character will be on the right and the high order Character on the left.

*)
(* read output adress to pointer *)
pt := ADR(DWORD_TO_STRH) + 8;
(* wirte the closing byte for the string *)
pt^:= 0;

(* write the 8 hex characters backwards *)
FOR i := 1 TO 8 DO;
	(* decrement the pointer *)
	pt := pt - 1;
	(* read the lowest order hex value *)
	temp := DWORD_TO_BYTE(in AND 16#0000000F);
	(* convert value to hex character *)
	IF temp <= 9 THEN temp := temp + 48; ELSE temp := temp + 55; END_IF;
	(* write character to output string *)
	PT^ := temp;
	(* shift in for nect hex character *)
	in := SHR(in,4);
END_FOR;


(* code beofre rev 1.2
FOR i := 1 TO 8 DO
	X := DWORD_TO_BYTE(in AND 2#1111);
	IF X <= 9 THEN X := X + 48; ELSE X := X + 55; END_IF;
	Cx := CHR(X);
	temp := CONCAT(Cx, temp);
	in := SHR(in,4);
END_FOR;
DWORD_TO_STRH := temp;
*)


(* revision history
hm		9.6.2007		rev 1.0		
	original version 

hm		11.9.2007		rev 1.1
	changed coding for compatibility with twincat, concat cannot support a function as an argument.

hm		15.12.2007		rev 1.2
	changed code for better performance
*)
END_FUNCTION

(* POU XTEST/Baustein Tests/esr_test, CFC *)
PROGRAM esr_test
VAR
	x1: ESR_collect;
	eout  : ARRAY[0..63] OF esr_data;
	x2: ESR_MON_B8;
	e0, e1, e2, e3, e4, e5, e6, e7: BOOL;
	dtime: DT;
	x3: ESR_MON_R4;
	r0, r1, r2, r3: REAL;
	x4: ESR_MON_X8;
	b0, b1, b2, b3, b4, b5, b6, b7: BYTE;
	m: BYTE;
	n: INT;
END_VAR
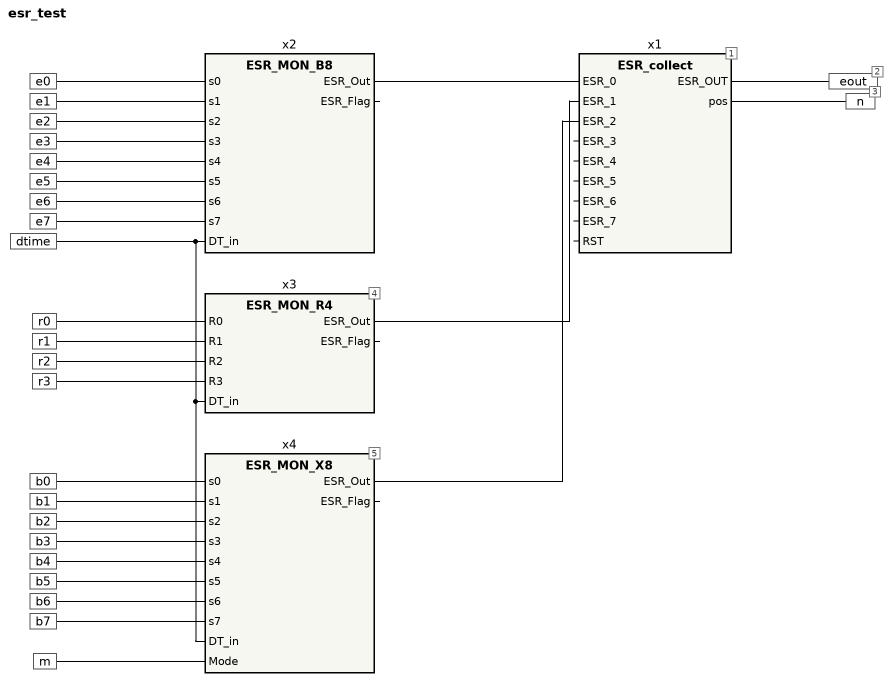
_CFC_ (* Continuous Function Chart, elements in execution order *)
#0 x2:ESR_MON_B8(s0: e0, s1: e1, s2: e2, s3: e3, s4: e4, s5: e5, s6: e6, s7: e7, DT_in: dtime, a0 := 'binär 0', a1 := 'binär 1', a2 := 'binär 2', a3 := 'binär 3', a4 := 'binär 4', a5 := 'binär 5', a6 := 'binär 6', a7 := 'binär 7')
#1 x1:ESR_collect(ESR_0: #0.ESR_Out, ESR_1: #4.ESR_Out, ESR_2: #5.ESR_Out, ESR_3: -, ESR_4: -, ESR_5: -, ESR_6: -, ESR_7: -, RST: -)
#2 eout <= #1.ESR_OUT
#3 n <= #1.pos
#4 x3:ESR_MON_R4(R0: r0, R1: r1, R2: r2, R3: r3, DT_in: dtime, a0 := 'real 0', a1 := 'real 1', a2 := 'real 2', a3 := 'real 3', s0 := 0.0, s1 := 0.1, s2 := 0.2, s3 := 0.3)
#5 x4:ESR_MON_X8(s0: b0, s1: b1, s2: b2, s3: b3, s4: b4, s5: b5, s6: b6, s7: b7, DT_in: dtime, Mode: m, a0 := 'status 0', a1 := 'status 1', a2 := 'status 2', a3 := 'status 3', a4 := 'status 4', a5 := 'status 5', a6 := 'status 6', a7 := 'status 7')
_END_CFC_
(* the same logic as Structured Text *)
x2(s0 := e0, s1 := e1, s2 := e2, s3 := e3, s4 := e4, s5 := e5, s6 := e6, s7 := e7, DT_in := dtime, a0 := 'binär 0', a1 := 'binär 1', a2 := 'binär 2', a3 := 'binär 3', a4 := 'binär 4', a5 := 'binär 5', a6 := 'binär 6', a7 := 'binär 7');
x1(ESR_0 := x2.ESR_Out, ESR_1 := x3.ESR_Out, ESR_2 := x4.ESR_Out);
eout := x1.ESR_OUT;
n := x1.pos;
x3(R0 := r0, R1 := r1, R2 := r2, R3 := r3, DT_in := dtime, a0 := 'real 0', a1 := 'real 1', a2 := 'real 2', a3 := 'real 3', s0 := 0.0, s1 := 0.1, s2 := 0.2, s3 := 0.3);
x4(s0 := b0, s1 := b1, s2 := b2, s3 := b3, s4 := b4, s5 := b5, s6 := b6, s7 := b7, DT_in := dtime, Mode := m, a0 := 'status 0', a1 := 'status 1', a2 := 'status 2', a3 := 'status 3', a4 := 'status 4', a5 := 'status 5', a6 := 'status 6', a7 := 'status 7');
END_PROGRAM

(* POU other/ESR_collect, ST *)
FUNCTION_BLOCK ESR_collect
VAR_INPUT
	ESR_0, ESR_1, ESR_2, ESR_3, ESR_4, ESR_5, ESR_6, ESR_7 : ARRAY [0..3] OF esr_data;
	RST : BOOL;
END_VAR
VAR_OUTPUT
	ESR_OUT : ARRAY[0..63] OF esr_data;
	pos : INT;
END_VAR
VAR CONSTANT
	max_in : INT := 3; (* maximum element of input variable *)
	max_out : INT := 63; (* maximum element of output array *)
END_VAR
VAR
	cnt : INT;
END_VAR

(*
version 1.0	26 jan 2007
programmer 	hugo
tested by		tobias

ESR_collect collects esr data from up to 8 esr_mon modules and stroes them in an output array.
the output pos will display the position of the last element in the array.
if the array will be full, the oldest element is overwritten.

*)
IF rst THEN
	pos := 0;
	FOR cnt := 0 TO 63 DO
		esr_out[cnt].typ := 0;
		esr_out[cnt].adress := '';
		esr_out[cnt].DS := DT#1970-1-1-00:00;
		esr_out[cnt].TS := T#0ms;
		esr_out[cnt].data[0] := 0;
		esr_out[cnt].data[1] := 0;
		esr_out[cnt].data[2] := 0;
		esr_out[cnt].data[3] := 0;
		esr_out[cnt].data[4] := 0;
		esr_out[cnt].data[5] := 0;
		esr_out[cnt].data[6] := 0;
		esr_out[cnt].data[7] := 0;
	END_FOR;
ELSE
	FOR cnt := 0 TO max_in DO
		IF esr_0[cnt].typ > 0 THEN
			esr_out[pos] := esr_0[cnt];
			pos := pos + 1;
			IF pos > max_out THEN pos := 0; END_IF;
		END_IF;
	END_FOR;
	FOR cnt := 0 TO max_in DO
		IF esr_1[cnt].typ > 0 THEN
			esr_out[pos] := esr_1[cnt];
			pos := pos + 1;
			IF pos > max_out THEN pos := 0; END_IF;
		END_IF;
	END_FOR;
	FOR cnt := 0 TO max_in DO
		IF esr_2[cnt].typ > 0 THEN
			esr_out[pos] := esr_2[cnt];
			pos := pos + 1;
			IF pos > max_out THEN pos := 0; END_IF;
		END_IF;
	END_FOR;
	FOR cnt := 0 TO max_in DO
		IF esr_3[cnt].typ > 0 THEN
			esr_out[pos] := esr_3[cnt];
			pos := pos + 1;
			IF pos > max_out THEN pos := 0; END_IF;
		END_IF;
	END_FOR;
	FOR cnt := 0 TO max_in DO
		IF esr_4[cnt].typ > 0 THEN
			esr_out[pos] := esr_4[cnt];
			pos := pos + 1;
			IF pos > max_out THEN pos := 0; END_IF;
		END_IF;
	END_FOR;
	FOR cnt := 0 TO max_in DO
		IF esr_5[cnt].typ > 0 THEN
			esr_out[pos] := esr_5[cnt];
			pos := pos + 1;
			IF pos > max_out THEN pos := 0; END_IF;
		END_IF;
	END_FOR;
	FOR cnt := 0 TO max_in DO
		IF esr_6[cnt].typ > 0 THEN
			esr_out[pos] := esr_6[cnt];
			pos := pos + 1;
			IF pos > max_out THEN pos := 0; END_IF;
		END_IF;
	END_FOR;
	FOR cnt := 0 TO max_in DO
		IF esr_7[cnt].typ > 0 THEN
			esr_out[pos] := esr_7[cnt];
			pos := pos + 1;
			IF pos > max_out THEN pos := 0; END_IF;
		END_IF;
	END_FOR;
END_IF;

(* revision history
hm	26.jan 2007		rev 1.0
	original version

hm	8. dec 2007		rev 1.1
	added reset input

*)
END_FUNCTION_BLOCK

(* POU other/ESR_MON_B8, ST *)
FUNCTION_BLOCK ESR_MON_B8
VAR_INPUT
	s0, s1, s2, s3, s4, s5, s6, s7 : BOOL;
	DT_in : DT;
END_VAR
VAR_INPUT CONSTANT
	a0, a1, a2, a3, a4, a5, a6, a7 : STRING(10);
END_VAR
VAR_OUTPUT
	ESR_Out: ARRAY [0..3] OF esr_data;
	ESR_Flag : BOOL;
END_VAR
VAR
	x0, x1, x2, x3, x4, x5, x6, x7 : BOOL;
	tx: TIME;
	cnt : INT;
END_VAR

(*
version 1.1	17 sep 2007
programmer 	hugo
tested by		tobias

ESR_mon_B8 monitores up to 8 binary inputs and reports changes with time stamd and adress label.
the module checks 8 inputs for a change and reports all changes with time and adress stamp to the output.
4 events maximum can be collected at once within the same cycle

*)
(* read system timer *)
tx := DWORD_TO_TIME(T_PLC_MS());

ESR_Flag := FALSE;
esr_out[3].typ := 0;
esr_out[2].typ := 0;
esr_out[1].typ := 0;
esr_out[0].typ := 0;
cnt := 0;

(* check if inputs have chaged and fill buffer *)
IF s0 <> X0 THEN
	IF s0 THEN esr_out[cnt].typ := 11; ELSE 	esr_out[cnt].typ := 10; END_IF;
	esr_out[cnt].adress := a0;
	esr_out[cnt].DS := DT_in;
	esr_out[cnt].TS := TX;
	X0 := S0;
	cnt := cnt + 1;
	esr_flag := TRUE;
END_IF;
IF s1 <> X1 THEN
	IF s1 THEN esr_out[cnt].typ := 11; ELSE 	esr_out[cnt].typ := 10; END_IF;
	esr_out[cnt].adress := a1;
	esr_out[cnt].DS := DT_in;
	esr_out[cnt].TS := TX;
	X1 := S1;
	cnt := cnt + 1;
	esr_flag := TRUE;
END_IF;
IF s2 <> X2 THEN
	IF s2 THEN esr_out[cnt].typ := 11; ELSE 	esr_out[cnt].typ := 10; END_IF;
	esr_out[cnt].adress := a2;
	esr_out[cnt].DS := DT_in;
	esr_out[cnt].TS := TX;
	X2 := S2;
	cnt := cnt + 1;
	esr_flag := TRUE;
END_IF;
IF s3 <> X3 THEN
	IF s3 THEN esr_out[cnt].typ := 11; ELSE 	esr_out[cnt].typ := 10; END_IF;
	esr_out[cnt].adress := a3;
	esr_out[cnt].DS := DT_in;
	esr_out[cnt].TS := TX;
	X3 := S3;
	cnt := cnt + 1;
	esr_flag := TRUE;
END_IF;
IF s4 <> X4 AND cnt < 4 THEN
	IF s4 THEN esr_out[cnt].typ := 11; ELSE 	esr_out[cnt].typ := 10; END_IF;
	esr_out[cnt].adress := a4;
	esr_out[cnt].DS := DT_in;
	esr_out[cnt].TS := TX;
	X4 := S4;
	cnt := cnt + 1;
	esr_flag := TRUE;
END_IF;
IF s5 <> X5  AND cnt < 4 THEN
	IF s5 THEN esr_out[cnt].typ := 11; ELSE 	esr_out[cnt].typ := 10; END_IF;
	esr_out[cnt].adress := a5;
	esr_out[cnt].DS := DT_in;
	esr_out[cnt].TS := TX;
	X5 := S5;
	cnt := cnt + 1;
	esr_flag := TRUE;
END_IF;
IF s6 <> X6  AND cnt < 4 THEN
	IF s6 THEN esr_out[cnt].typ := 11; ELSE 	esr_out[cnt].typ := 10; END_IF;
	esr_out[cnt].adress := a6;
	esr_out[cnt].DS := DT_in;
	esr_out[cnt].TS := TX;
	X6 := S6;
	cnt := cnt + 1;
	esr_flag := TRUE;
END_IF;
IF s7 <> X7  AND cnt < 4 THEN
	IF s7 THEN esr_out[cnt].typ := 11; ELSE 	esr_out[cnt].typ := 10; END_IF;
	esr_out[cnt].adress := a7;
	esr_out[cnt].DS := DT_in;
	esr_out[cnt].TS := TX;
	X7 := S7;
	cnt := cnt + 1;
	esr_flag := TRUE;
END_IF;

(* revision history
hm	26. jan 2007		rev 1.0
	original version

hm	17. sep 2007	rev 1.1
	replaced time() with T_PLC_MS() for compatibility reasons
	
*)
END_FUNCTION_BLOCK

(* POU other/ESR_MON_R4, ST *)
FUNCTION_BLOCK ESR_MON_R4
VAR_INPUT
	R0, R1, R2, R3 : REAL;
	DT_in : DT;
END_VAR
VAR_INPUT CONSTANT
	a0, a1, a2, a3 : STRING(10);
	s0, s1, s2, s3 : REAL;
END_VAR
VAR_OUTPUT
	ESR_Out: ARRAY [0..3] OF esr_data;
	ESR_Flag : BOOL;
END_VAR
VAR
	p0, p1, p2, p3 : POINTER TO DWORD;
	x0, x1, x2, x3 : REAL;
	tx: TIME;
	cnt : INT;
END_VAR

(*
version 1.2 8 dec 2007
programmer 	hugo
tested by		tobias

ESR_mon_R4 monitores up to 4 Real inputs and reports changes with time stamd and adress label.
the module checks 4 inputs for a change of more than the specified sensitivity S and reports all changes with time and adress stamp to the output.

*)
(* read system timer *)
tx := DWORD_TO_TIME(T_PLC_MS());
P0 := ADR(R0);
P1 := ADR(R1);
P2 := ADR(R2);
P3 := ADR(R3);

ESR_Flag := FALSE;
esr_out[3].typ := 0;
esr_out[2].typ := 0;
esr_out[1].typ := 0;
esr_out[0].typ := 0;
cnt := 0;

(* check if inputs have chaged and fill buffer *)
IF differ(R0,  X0, S0) THEN
	esr_out[cnt].typ := 20;
	esr_out[cnt].adress := a0;
	esr_out[cnt].DS := DT_in;
	esr_out[cnt].TS := TX;
	esr_out[cnt].data[0] := Byte_of_Dword(REAL_TO_DWORD(P0^),0);
	esr_out[cnt].data[1] := Byte_of_Dword(REAL_TO_DWORD(P0^),1);
	esr_out[cnt].data[2] := Byte_of_Dword(REAL_TO_DWORD(P0^),2);
	esr_out[cnt].data[3] := Byte_of_Dword(REAL_TO_DWORD(P0^),3);
	X0 := R0;
	cnt := cnt + 1;
	esr_flag := TRUE;
END_IF;
IF differ(R1,  X1, S1) THEN
	esr_out[cnt].typ := 20;
	esr_out[cnt].adress := a1;
	esr_out[cnt].DS := DT_in;
	esr_out[cnt].TS := TX;
	esr_out[cnt].data[0] := Byte_of_Dword(REAL_TO_DWORD(P1^),0);
	esr_out[cnt].data[1] := Byte_of_Dword(REAL_TO_DWORD(P1^),1);
	esr_out[cnt].data[2] := Byte_of_Dword(REAL_TO_DWORD(P1^),2);
	esr_out[cnt].data[3] := Byte_of_Dword(REAL_TO_DWORD(P1^),3);
	X1 := R1;
	cnt := cnt + 1;
	esr_flag := TRUE;
END_IF;
IF differ(R2,  X2, S2) THEN
	esr_out[cnt].typ := 20;
	esr_out[cnt].adress := a2;
	esr_out[cnt].DS := DT_in;
	esr_out[cnt].TS := TX;
	esr_out[cnt].data[0] := Byte_of_Dword(REAL_TO_DWORD(P2^),0);
	esr_out[cnt].data[1] := Byte_of_Dword(REAL_TO_DWORD(P2^),1);
	esr_out[cnt].data[2] := Byte_of_Dword(REAL_TO_DWORD(P2^),2);
	esr_out[cnt].data[3] := Byte_of_Dword(REAL_TO_DWORD(P2^),3);
	X2 := R2;
	cnt := cnt + 1;
	esr_flag := TRUE;
END_IF;
IF differ(R3,  X3, S3) THEN
	esr_out[cnt].typ := 20;
	esr_out[cnt].adress := a3;
	esr_out[cnt].DS := DT_in;
	esr_out[cnt].TS := TX;
	esr_out[cnt].data[0] := Byte_of_Dword(REAL_TO_DWORD(P3^),0);
	esr_out[cnt].data[1] := Byte_of_Dword(REAL_TO_DWORD(P3^),1);
	esr_out[cnt].data[2] := Byte_of_Dword(REAL_TO_DWORD(P3^),2);
	esr_out[cnt].data[3] := Byte_of_Dword(REAL_TO_DWORD(P3^),3);
	X3 := R3;
	cnt := cnt + 1;
	esr_flag := TRUE;
END_IF;


(* revision history
hm	26. jan 2007	rev 1.0
	original version

hm	17. sep 2007	rev 1.1
	replaced time() with T_PLC_MS() for compatibility reasons

hm	8 dec 2007		rev 1.2
	corrected an error while esr typ would not be set
*)
END_FUNCTION_BLOCK

(* POU mathematical/differ, ST *)
FUNCTION differ : BOOL
VAR_INPUT
	in1 : REAL;
	in2 : REAL;
	X : REAL;
END_VAR
VAR
END_VAR

(*
version 1.0	8 oct 2006
programmer 	hugo
tested by		tobias

this function checks if in1 differs more then x from in2
the output is true if in1 < in2 - x or in1 > in2 + X
*)
differ := in1 < in2 - X OR in1 > in2 + X;
END_FUNCTION

(* POU Logic/gate logic/Byte_of_Dword, ST *)
FUNCTION Byte_of_Dword : BYTE
VAR_INPUT
	in : DWORD;
	N : BYTE;
END_VAR
VAR
END_VAR

(*
version 1.1	2 jan 2008
programmer 	hugo
tested by		tobias

this function extracts a single byte from the nth position from right (right is lowest byte) 
the lower byte (starting with Bit0 from in) is selected with N=0.
*)
Byte_of_Dword := DWORD_TO_BYTE(SHR(in,n*8));

(* revision history
hm	17. jan 2007	rev 1.0
	original version

hm	2. jan 2008		rev 1.1
	improved performance

*)
END_FUNCTION

(* POU other/ESR_MON_X8, ST *)
FUNCTION_BLOCK ESR_MON_X8
VAR_INPUT
	s0, s1, s2, s3, s4, s5, s6, s7 : BYTE;
	DT_in : DT;
	Mode : BYTE := 3;
END_VAR
VAR_INPUT CONSTANT
	a0, a1, a2, a3, a4, a5, a6, a7 : STRING(10);
END_VAR
VAR_OUTPUT
	ESR_Out: ARRAY [0..3] OF esr_data;
	ESR_Flag : BOOL;
END_VAR
VAR
	x0, x1, x2, x3, x4, x5, x6, x7 : BYTE;
	tx: TIME;
	cnt : INT;
END_VAR

(*
version 1.1	17 sep 2007
programmer 	hugo
tested by		tobias

ESR_MON_X8 is a status and error collector.
the module checks 8 status inputs for a change and reports up to 4 input changes with time and adress stamp to the output.
the mode can be 
1 for error only
2 for error and status
3 for error, status and debug
the adress label of the 8 inputs can be configured individually.
*)
(* read system timer *)
tx := DWORD_TO_TIME(T_PLC_MS());

ESR_Flag := FALSE;
esr_out[3].typ := 0;
esr_out[2].typ := 0;
esr_out[1].typ := 0;
esr_out[0].typ := 0;
cnt := 0;

(* check if inputs have chaged and fill buffer *)
IF s0 <> X0 AND ((s0 < 100) OR (S0 > 99 AND S0 < 200 AND mode >= 2) OR (S0 > 199 AND mode = 3)) THEN
	esr_out[cnt] := status_to_ESR(s0, a0, DT_in, TX);
	X0 := S0;
	cnt := cnt + 1;
	esr_flag := TRUE;
END_IF;
IF s1 <> X1 AND ((s1 < 100) OR (S1 > 99 AND S1 < 200 AND mode >= 2) OR (S1 > 199 AND mode = 3)) THEN
	esr_out[cnt] := status_to_ESR(s1, a1, DT_in, TX);
	X1 := S1;
	cnt := cnt + 1;
	esr_flag := TRUE;
END_IF;
IF s2 <> X2 AND ((s2 < 100) OR (S2 > 99 AND S2 < 200 AND mode >= 2) OR (S2 > 199 AND mode = 3)) THEN
	esr_out[cnt] := status_to_ESR(s2, a2, DT_in, TX);
	X2 := S2;
	cnt := cnt + 1;
	esr_flag := TRUE;
END_IF;
IF s3 <> X3 AND ((s3 < 100) OR (S3 > 99 AND S3 < 200 AND mode >= 2) OR (S3 > 199 AND mode = 3)) THEN
	esr_out[cnt] := status_to_ESR(s3, a3, DT_in, TX);
	X3 := S3;
	cnt := cnt + 1;
	esr_flag := TRUE;
END_IF;
IF cnt < 4 AND s4 <> X4 AND ((s4 < 100) OR (S4 > 99 AND S4 < 200 AND mode >= 2) OR (S4 > 199 AND mode = 3)) THEN
	esr_out[cnt] := status_to_ESR(s4, a4, DT_in, TX);
	X4 := S4;
	cnt := cnt + 1;
	esr_flag := TRUE;
END_IF;
IF cnt < 4 AND s5 <> X5 AND ((s5 < 100) OR (S5 > 99 AND S5 < 200 AND mode >= 2) OR (S5 > 199 AND mode = 3)) THEN
	esr_out[cnt] := status_to_ESR(s5, a5, DT_in, TX);
	X5 := S5;
	cnt := cnt + 1;
	esr_flag := TRUE;
END_IF;
IF cnt < 4 AND s6 <> X6 AND ((s6 < 100) OR (S6 > 99 AND S6 < 200 AND mode >= 2) OR (S6 > 199 AND mode = 3)) THEN
	esr_out[cnt] := status_to_ESR(s6, a6, DT_in, TX);
	X6 := S6;
	cnt := cnt + 1;
	esr_flag := TRUE;
END_IF;
IF cnt < 4 AND s7 <> X7 AND ((s7 < 100) OR (S7 > 99 AND S7 < 200 AND mode >= 2) OR (S7 > 199 AND mode = 3)) THEN
	esr_out[cnt] := status_to_ESR(s7, a7, DT_in, TX);
	X7 := S7;
	cnt := cnt + 1;
	esr_flag := TRUE;
END_IF;


(* revision history
hm	26. jan 2007		rev 1.0
	original version

hm	17. sep 2007	rev 1.1
	replaced time() with T_PLC_MS() for compatibility reasons
	
*)
END_FUNCTION_BLOCK

(* POU other/status_to_ESR, ST *)
FUNCTION status_to_ESR : esr_data
VAR_INPUT
	status : BYTE;
	adress : STRING(10);
	DT_in : DT;
	TS : TIME;
END_VAR
VAR
END_VAR

(*
version 1.0	6 oct 2006
programmer 	hugo
tested by		tobias

status_to_esr creates esr data from a status byte.

*)
IF status < 100 THEN
	status_to_ESR.typ := 1;
ELSIF status < 200 THEN
	status_to_ESR.typ := 2;
ELSE
	status_to_ESR.typ := 3;
END_IF;
status_to_ESR.adress:= adress;
status_to_ESR.DS := DT_in;
status_to_ESR.TS := TS;
status_to_ESR.data[0] := status;
END_FUNCTION

(* POU XTEST/Baustein Tests/gen_rdt_test, CFC *)
PROGRAM gen_rdt_test
VAR
	x1: GEN_RDT;
	out: BOOL;
	start: BOOL;
	x2: TP;
	o2: BOOL;
END_VAR
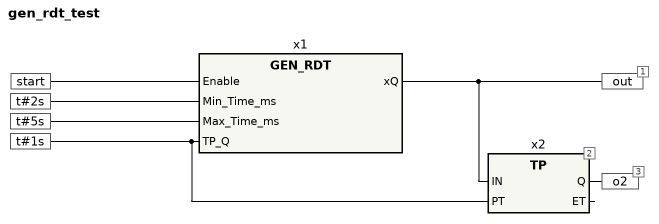
_CFC_ (* Continuous Function Chart, elements in execution order *)
#0 x1:GEN_RDT(Enable: start, Min_Time_ms: t#2s, Max_Time_ms: t#5s, TP_Q: t#1s)
#1 out <= #0.xQ
#2 x2:TP(IN: #0.xQ, PT: t#1s)
#3 o2 <= #2.Q
_END_CFC_
(* the same logic as Structured Text *)
x1(Enable := start, Min_Time_ms := t#2s, Max_Time_ms := t#5s, TP_Q := t#1s);
out := x1.xQ;
x2(IN := x1.xQ, PT := t#1s);
o2 := x2.Q;
END_PROGRAM

(* POU engineering/signal generators/GEN_RDT, ST *)
FUNCTION_BLOCK GEN_RDT

VAR_INPUT
		 Enable		 	: BOOL := TRUE ;
		 Min_Time_ms	: TIME := t#1s ; (* min Taktzeit *)
		 Max_Time_ms	: TIME := t#1.2s ; (* Max Taktzeit *)
		 TP_Q		 		: TIME := t#100ms ; (* Zeit Ausgang auf TRUE *)
END_VAR
VAR_OUTPUT
		 xQ		 : BOOL ;
END_VAR
VAR
(* Taktgenerator Simulation *)
		 tonRDMTimer		: TON ; (* Zeitbaustein Taktgenerator *)
		 tof_xQ		 		: TOF ; (* Ausschaltverzögerung Taktgenerator *)
		 tRDMTime		: TIME ; (* Sollzeit *)
		 rRDMTime		: REAL ; (* Zufalswert Timer *)
END_VAR

(*
version 1.2	1 nov 2007
programmer 	J. Schohaus
tested by		Hugo

RDMT generates a defined pulse with pulse width TP_Q at random times. the random time will be defined with an minimum and maximum time.

*)


(*
FUNCTION_BLOCK RDMTimer
###############################################################################
		 Ersteller / author :		 		 		 		 		 J.Schohaus
		 Datum / date:		 		 		 		 		 		 13.07.2007
###############################################################################
		 Änderungen / Datum / Ersteller :		 		 		 		 		 		 		 		 		 		 		 		 		 		 		 
		 moditication / date / author :		 		 
###############################################################################
		 Verwendete Bibliotheken		 ( * werden im Baustein nicht benötigt )
		 		 		 		 Oscat.lib
###############################################################################
Beschreibung:
*)
tonRDMTimer ( IN:= Enable , PT:= tRDMTime );
tof_xQ ( IN:= tonRDMTimer.Q , PT:= TP_Q );
XQ := tof_xq.Q;
IF tonRDMTimer.Q THEN
		 xQ := TRUE ;
		 rRDMTime := RDM ( last:= rRDMTime ) ;
		 tRDMTime := REAL_TO_TIME ( rRDMTime * TIME_TO_DINT( Max_Time_ms - Min_Time_ms ) + TIME_TO_DINT(Min_Time_ms )) ;
		 tonRDMTimer ( IN:= FALSE );
END_IF;

(* revision history
J. Schohaus	19. nov 2007		rev 1.0
	origial version

*)
END_FUNCTION_BLOCK

(* POU mathematical/RDM, ST *)
FUNCTION RDM : REAL
VAR_INPUT
	last : REAL;
END_VAR
VAR
	tn : DWORD;
	tc : INT;
END_VAR


(*
version 1.4	2 feb 2008
programmer 	hugo
tested by	tobias

this function calculates a pseudo random number
to generate the number it reads the sps timer and calculates a random number between 0 and 1:
in order to use rdm more then once within one sps cycle it need to be called with different seed numbers LAST.

*)
tn := T_PLC_MS();
tc := Bit_Count(tn);
tn.31 := tn.2;
tn.30 := tn.5;
tn.29 := tn.4;
tn.28 := tn.1;
tn.27 := tn.0;
tn.26 := tn.7;
tn.25 := tn.6;
tn.24 := tn.3;
tn := ROL(tn,Bit_Count(tn)) OR 16#80000001;
tn := tn MOD 71474513 + tc + 77;
RDM := fract(DWORD_TO_REAL(tn) / 10000000 * (e-last));


(*
pt := ADR(temp);
pt^ := (T_PLC_MS() AND 16#007FFFFF) OR 16#3D000000;
RDM := fract(modR(temp*e+pi1, PI1-last) + modR(temp*PI1+e + last,e-last));
*)

(* revision history
hm		16. jan 2007		rev 1.0
	original version

hm		11. nov 2007		rev 1.1
	changed time() into t_plc_ms()

hm		20. nov 2007		rev 1.2
	changed code of temp calculation to avoid overflow in modr due to resuclt would not fit DINT for high timeer values

hm		5. jan 2008			rev 1.3
	changed calculation of temp to avoid problem with high values of t_plc_ms

hm		2. feb 2008			rev 1.4
	changed algorithm to avoind non iec functions and guarantee more randomness
*)
END_FUNCTION

(* POU Logic/gate logic/Bit_Count, ST *)
FUNCTION Bit_Count : INT
VAR_INPUT
	IN : DWORD;
END_VAR
VAR
END_VAR

(*
version 1.1	10 sep 2007
programmer 	hugo
tested by		tobias

BIT_COUNT counts the amount True of bits in a dword.
for exabple: bit_count(3) returns 2 because two bits (bits 0 and 1) are true and all others are false. 

*)
WHILE in > 0 DO
	IF in.0 THEN Bit_Count := Bit_Count +1; END_IF;
	in := SHR(in,1);
END_WHILE;

(* revision history
5.7.2007	rev 1.0		original version

10.9.2007	rev 1.1		hm
	changed algorithm for better performace
	the execution time has reduced by a factor of 5
	deleted unused variable temp
*)
END_FUNCTION

(* POU mathematical/fract, ST *)
FUNCTION fract : REAL
VAR_INPUT
	input : REAL;
END_VAR
VAR
END_VAR
VAR
END_VAR

(*
version 1.0	4 aug 2006
programmer 	hugo
tested by		tobias

this function returns the fraction of a real number
fract(3.14) = 0.14

*)
fract := input - TRUNC(input);
END_FUNCTION

(* POU XTEST/Baustein Tests/heat_meter_test, CFC *)
PROGRAM heat_meter_test
VAR
	kj : REAL;
	x1: heat_meter;
	run: BOOL;
	rst: BOOL;
	den: REAL;
	ent: REAL;
	x2: TP;
END_VAR
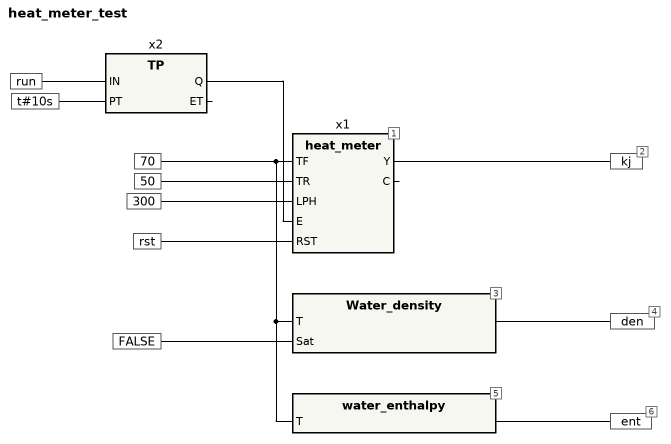
_CFC_ (* Continuous Function Chart, elements in execution order *)
#0 x2:TP(IN: run, PT: t#10s)
#1 x1:heat_meter(TF: 70, TR: 50, LPH: 300, E: #0.Q, RST: rst, Pulse_Mode := TRUE)
#2 kj <= #1.Y
#3 Water_density(T: 70, Sat: FALSE)
#4 den <= #3
#5 water_enthalpy(T: 70)
#6 ent <= #5
_END_CFC_
END_PROGRAM

(* POU Building/HLK/heat_meter, ST *)
FUNCTION_BLOCK heat_meter
VAR_INPUT
	TF, TR : REAL;
	LPH : REAL;
	E : BOOL;
	RST : BOOL;
END_VAR
VAR_INPUT CONSTANT
	CP : REAL;
	Density : REAL;
	Content : REAL;
	Pulse_Mode : BOOL;
	Return_meter : BOOL;
	AVG_time : TIME := T#5s;
END_VAR
VAR_OUTPUT
	Y : REAL;
	C : REAL;
END_VAR
VAR
	tx, last : DWORD;
	int1 : FT_INT;
	edge : BOOL;
	X: REAL;
	init: BOOL;
	Y_last: REAL;
END_VAR

(*
version 1.1	25 dec 2007
programmer 	hugo
tested by		tobias

Heat meter measures the heat transfer of water of a mixture of water and another component.
The inputs are foreward temperature and reverse temperature.
the additional component is specified with its parameters density, Specific heat capacity and content in %.
an input e anables the measurement while it can be configured to be based on X liters / pulse or in liters / hour.
the output is in Joule.

*)
IF rst THEN
	int1(rst := TRUE);
	int1.rst := FALSE;
	C := 0;
	Y := 0;
ELSIF pulse_mode AND e AND NOT edge THEN
	IF return_meter THEN
		X := (Water_density(TR, FALSE) * (water_enthalpy(TF) - water_enthalpy(TR)) * (1-content) + CP * Density * content*(TF-TR));
	ELSE
		X := (Water_density(TF, FALSE) * (water_enthalpy(TF) - water_enthalpy(TR)) * (1-content) + CP * Density * content*(TF-TR));
	END_IF;
	Y := Y + X * LPH;
	edge := e;
ELSIF NOT pulse_mode AND e THEN
	IF return_meter THEN
		X := (Water_density(TR, FALSE) * (water_enthalpy(TF) - water_enthalpy(TR)) * (1-content) + CP * Density * content*(TF-TR));
	ELSE
		X := (Water_density(TF, FALSE) * (water_enthalpy(TF) - water_enthalpy(TR)) * (1-content) + CP * Density * content*(TF-TR));
	END_IF;
	int1(in := X * LPH / 3600.0, out_min := 0, out_max := 3E38);
	Y := int1.Out;
END_IF;

(* read system_time *)
tx := T_PLC_MS();

(* only init at startup necessary *)
IF NOT init THEN
	init := TRUE;
	last := tx;
END_IF;

(* calculate the current consumption *)
IF (tx - last >= TIME_TO_DWORD(AVG_TIME)) AND (avg_time > T#0s) THEN
	last := tx;
	C := (Y - Y_last) * 3.6/TIME_TO_DWORD(AVG_TIME);
	Y_last := Y;
END_IF;



(* revision history
hm		16.11.2007	rev 1.0
	original version

hm		24.12.2007	rev 1.1
	added config variable return_meter
	added output C for current consumption
*)
END_FUNCTION_BLOCK

(* POU Building/HLK/Water_density, ST *)
FUNCTION Water_density : REAL
VAR_INPUT
	T : REAL;
	Sat : BOOL;
END_VAR
VAR CONSTANT
	a0 : REAL := 999.83952;
	a1 : REAL := 16.952577;
	a2 : REAL := -7.9905127E-3;
	a3 : REAL := -4.6241757E-5;
	a4 : REAL := 1.0584601E-7;
	a5 : REAL := -2.8103006E-10;
	b  : REAL := 0.0168872;
END_VAR
VAR
	T2: REAL;
	T4: REAL;
END_VAR


(*
version 1.1	2 dec 2007
programmer 	hugo
tested by		tobias

this function calculates the water density for air free water between 0 and 100 deg C
while sat is false the denisty is calculated for air free water and when sat = true
the calculation is performed for water saturated with air.

*)
T2 := T * T;
T4 := T2 * T2;

(* original code changed for performance
Water_density := (a0 + a1*T + a2*EXPT(T,2) + a3*EXPT(t,3) + a4*EXPT(t,4) + a5*EXPT(t,5)) / (1 + b*T);
*)
Water_density := (a0 + a1*T + a2*T2 + a3*T2*T + a4*T4 + a5*T4*T) / (1 + b*T);

IF sat THEN Water_density := Water_density - 0.004612 + 0.000106 * T; END_IF;


(* revision history

hm	13.9.2007		rev 1.0
	original version

hm	2.12.2007		rev 1.1
	changed code for better performance
*)

(*
    °C - die Celsius-Temperatur in Grad Celsius
    v – das spezifische Volumen in Kubikdezimeter je Kilogramm dm³/kg
    h – die spezifische Enthalpie in Kilojoule je Kilogramm 	kJ/kg
    u – die spezifische Innere Energie in Kilojoule je Kilogramm 	kJ/kg
    s – die spezifische Entropie in Kilojoule je Kilogramm mal Kelvin 	kJ/(kg·K)
    cp - die spezifische Wärmekapazität bei konstantem Druck in Kilojoule je Kilogramm mal Kelvin 	kJ/(kg·K)
    Y – Volumenausdehnungskoeffizient in 10-3 durch Kelvin  10-3/K
    L – Wärmeleitfähigkeit in Milliwatt je Meter mal Kelvin  mW / (m·K) 
    n – Viskosität in Mikropascal mal Sekunde uPa·s 	
    s ? – Oberflächenspannung in Millinewton je Meter  mN/m


°C 		v 				h 			u 		s 			cp 		Y 		L		n		s	
-20		1,006580	
0 		1,000160 		0,06 		-0,04 	-0,0001 	4,228 	-0,080 	561,0 	1792 	75,65
4		1,000028
5 		1,0000 		21,1 		21,0 	0,076 		4,200 	0,011 	570,6 	1518 	74,95
10 		1,0003 		42,1 		42,0 	0,151 		4,188 	0,087 	580,0 	1306 	74,22
15 		1,0009 		63,0 		62,9 	0,224 		4,184 	0,152 	589,4 	1137 	73,49
20 		1,001797 		83,9 		83,8 	0,296 		4,183 	0,209 	598,4 	1001 	72,74
25 		1,0029 		104,8 		104,7 	0,367 		4,183 	0,259 	607,2 	890,4 	71,98
30 		1,0044 		125,8 		125,7 	0,437 		4,183 	0,305 	615,5 	797,7 	71,20
35 		1,0060 		146,7 		146,6 	0,505 		4,183 	0,347 	623,3 	719,6 	70,41
40 		1,007842 		167,58 	167,5 	0,572 		4,182 	0,386 	630,6 	653,3 	69,60
45 		1,0099 		188,5 		188,4 	0,638 		4,182 	0,423 	637,3 	596,3 	68,78
50 		1,0121 		209,4 		209,3 	0,704 		4,181 	0,457 	643,6 	547,1 	67,95
60 		1,017089 		251,2 		251,1 	0,831 		4,183 	0,522 	654,4 	466,6 	66,24
70 		1,0227 		293,1 		293,0 	0,955 		4,187 	0,583 	663,1 	404,1 	64,49
80 		1,029027 		335,0 		334,9 	1,075 		4,194 	0,640 	670,0 	354,5 	62,68
90 		1,0359 		377,0 		376,9 	1,193 		4,204 	0,696 	675,3 	314,6 	60,82
99,63 	1,0431 		417,5 		417,4 	1,303 		4,217 	0,748 	679,0 	283,0 	58,99
100	1,043453		419,1

Stoffdaten von Wasser Quelle Wickipedia

*)
END_FUNCTION

(* POU Building/HLK/water_enthalpy, ST *)
FUNCTION water_enthalpy : REAL
VAR_INPUT
	T : REAL;
END_VAR
VAR
	Pts : INT := 11;
	data : ARRAY[1..20, 0..1] OF REAL := 0,0.06, 10,42.1, 20,83.9, 30,125.8, 40,167.58, 50,209.4, 60,251.2, 70,293.1, 80,335.0, 90, 377.0, 100,419.1 ;
END_VAR

(*
version 1.0	29 oct 2007
programmer 	hugo
tested by		tobias

water_enthalpy calculates the enthalpy of liquid water from 0..100 °C 

*)
water_enthalpy := LINEAR_INT(T, Data, Pts);


(* revision history

hm	29.10.2007	rev 1.0
	original version

*)

(*
    °C - die Celsius-Temperatur in Grad Celsius
    v – das spezifische Volumen in Kubikdezimeter je Kilogramm dm³/kg
    h – die spezifische Enthalpie in Kilojoule je Kilogramm 	kJ/kg
    u – die spezifische Innere Energie in Kilojoule je Kilogramm 	kJ/kg
    s – die spezifische Entropie in Kilojoule je Kilogramm mal Kelvin 	kJ/(kg·K)
    cp - die spezifische Wärmekapazität bei konstantem Druck in Kilojoule je Kilogramm mal Kelvin 	kJ/(kg·K)
    Y – Volumenausdehnungskoeffizient in 10-3 durch Kelvin  10-3/K
    L – Wärmeleitfähigkeit in Milliwatt je Meter mal Kelvin  mW / (m·K) 
    n – Viskosität in Mikropascal mal Sekunde uPa·s 	
    s ? – Oberflächenspannung in Millinewton je Meter  mN/m


°C 		v 				h 			u 		s 			cp 		Y 		L		n		s	
-20		1,006580	
0 		1,000160 		0,06 		-0,04 	-0,0001 	4,228 	-0,080 	561,0 	1792 	75,65
4		1,000028
5 		1,0000 		21,1 		21,0 	0,076 		4,200 	0,011 	570,6 	1518 	74,95
10 		1,0003 		42,1 		42,0 	0,151 		4,188 	0,087 	580,0 	1306 	74,22
15 		1,0009 		63,0 		62,9 	0,224 		4,184 	0,152 	589,4 	1137 	73,49
20 		1,001797 		83,9 		83,8 	0,296 		4,183 	0,209 	598,4 	1001 	72,74
25 		1,0029 		104,8 		104,7 	0,367 		4,183 	0,259 	607,2 	890,4 	71,98
30 		1,0044 		125,8 		125,7 	0,437 		4,183 	0,305 	615,5 	797,7 	71,20
35 		1,0060 		146,7 		146,6 	0,505 		4,183 	0,347 	623,3 	719,6 	70,41
40 		1,007842 		167,58 	167,5 	0,572 		4,182 	0,386 	630,6 	653,3 	69,60
45 		1,0099 		188,5 		188,4 	0,638 		4,182 	0,423 	637,3 	596,3 	68,78
50 		1,0121 		209,4 		209,3 	0,704 		4,181 	0,457 	643,6 	547,1 	67,95
60 		1,017089 		251,2 		251,1 	0,831 		4,183 	0,522 	654,4 	466,6 	66,24
70 		1,0227 		293,1 		293,0 	0,955 		4,187 	0,583 	663,1 	404,1 	64,49
80 		1,029027 		335,0 		334,9 	1,075 		4,194 	0,640 	670,0 	354,5 	62,68
90 		1,0359 		377,0 		376,9 	1,193 		4,204 	0,696 	675,3 	314,6 	60,82
99,63 	1,0431 		417,5 		417,4 	1,303 		4,217 	0,748 	679,0 	283,0 	58,99
100	1,043453		419,1

Stoffdaten von Wasser Quelle Wickipedia

Wasser hat unter Normaldruck seine größte Dichte von 1000 Kilogramm pro Kubikmeter bei 3,98 °C und zeigt damit eine Dichteanomalie. 
Diese besteht darin, dass sich Wasser unterhalb von 3,98 °C bei weiterer Temperaturverringerung, auch beim Wechsel zum festen 
Aggregatzustand, wieder ausdehnt, was man nur von wenigen Stoffen kennt. Die derzeit genauesten publizierten Werte für die maximale 
Dichte liegen bei (999,974950 ± 0,00084) kg/m³ und bei (3,983 ± 0,00067) °C für die Temperatur, bei der dieser Wert erreicht wird. 
Die Werte stellen einen Mittelwert der von verschiedenen physikalischen Instituten veröffentlichten Zahlen dar (Stand 2001).

Die Berechnung der Dichte von luftfreiem Wasser DLF in Abhängigkeit von der Temperatur T ([T] = °C) kann mit Hilfe der folgenden 
Virialgleichung erfolgen:
: \frac{D_{\rm LF}}{\rm g/l} = \frac{a_0 + a_1 T + a_2 T^2 + a_3 T^3 + a_4 T^4 + a_5 T^5}{1 + b T}.
mit den Koeffizienten: a0 = 999,83952; a1 = 16,952577 (°C)-1; a2 = -7,9905127·10-3 (°C)-2; a3 = -4,6241757·10-5 (°C)-3; 
a4 = 1,0584601·10-7 (°C)-4; a5 = -2,8103006·10-10 (°C)-5 und b = 0,0168872. 
Für die Berechnung der Dichte von luftgesättigtem Wasser korrigiert man den Wert nach 
DLG/(g/l) = DLF/(g/l) - 0,004612 + 0,000106 (°C)-1·T. (Quelle: PTB-Mitteilungen 100/3-90)

*)
END_FUNCTION

(* POU mathematical/functions/LINEAR_INT, ST *)
FUNCTION LINEAR_INT : REAL
VAR_INPUT
	X : REAL;
	XY : ARRAY[1..20,0..1] OF REAL;
	Pts : INT;
END_VAR
VAR
	i : INT;
END_VAR

(*
	version 1.1	27 dec 2007
	programmer 	oscat
	tested BY		oscat

LINEAR_INT calculates an output based on a linear interpolation of up to 20 coordinates given in an array
the input coordinates have to start at the lowest array position and must be sorted ba ascending X values.

*)
(*make sure n is bound within the array size *)
pts := MIN(pts,20);

(* calculate the linear segement interpolation *)
i := 2;
(* search for segment and calculate output
	below and above the defined segments we interpolate the last segment *)
WHILE (i < pts) AND (XY[i,0] < X) DO
	i := i + 1;
END_WHILE;

(* calculate the output value on the corresponding segment coordinates *)
LINEAR_INT := ((XY[i,1] - XY[i-1,1]) * X - XY[i,1] * XY[i-1,0] + XY[i-1,1] * XY[i,0]) / (XY[i,0] - XY[i-1,0]);

(* revision history
hm	7. oct 2007		rev 1.0
	original version

hm	27 dec 2007		rev 1.1
	changed code for better performance
*)
END_FUNCTION

(* POU XTEST/Baustein Tests/holiday_test, CFC *)
PROGRAM holiday_test
VAR
	x1: holiday;
	dtin: DATE;
	hol: BOOL;
	nameh: STRING;
END_VAR
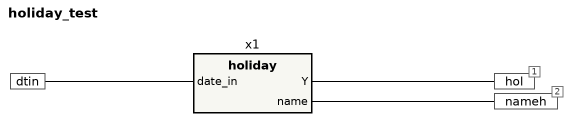
_CFC_ (* Continuous Function Chart, elements in execution order *)
#0 x1:holiday(date_in: dtin)
#1 hol <= #0.Y
#2 nameh <= #0.name
_END_CFC_
(* the same logic as Structured Text *)
x1(date_in := dtin);
hol := x1.Y;
nameh := x1.name;
END_PROGRAM

(* POU Time&Date/holiday, ST *)
FUNCTION_BLOCK holiday
VAR_INPUT
	date_in : DATE;
END_VAR
VAR_INPUT CONSTANT
	size : INT := 24;
	feiertag : ARRAY [0..24] OF STRING(27) := 'Neujahr', 'Heilig Drei Könige', 'Karfreitag', 'Ostersonntag', 'Ostermontag', 'Tag der Arbeit',
	'Christi Himmelfahrt', 'Pfingstsonntag', 'Pfingstmontag', 'Fronleichnam', 'Augsburger Friedensfest', 'Maria Himmelfahrt',
	'Tag der Deutschen Einheit', 'Reformationstag', 'Allerheiligen', 'Buss und Bettag', '1. Weihnachtstag', '2. Weihnachtstag';
	f_day : ARRAY [0..24] OF SINT := 1, 6, -2, 0, 1, 1, 39, 49, 50 , 60, 8, 15, 3, 31, 1, 23, 25, 26;
	f_month : ARRAY [0..24] OF SINT := 1, 1, 0, 0, 0, 5, 0, 0, 0, 0, 8, 8, 10, 10, 11, 11, 12, 12;
	(* if month = 0 then F_day is the offset in days from easter *)
	f_use : ARRAY [0..24] OF SINT := 1,1,1,1,1,1,1,1,1,1,0,1,1,0,1,0,1,1;
	(* 0 = not used, 1 = used, -1..-7 menas the weekday before the specified date example -3 means wednesday before 23.11 *)
	Friday : BOOL := FALSE;
	Saturday : BOOL := FALSE;
	Sunday : BOOL := FALSE;
END_VAR
VAR_OUTPUT
	Y : BOOL;
	name : STRING(20);
END_VAR
VAR
	last_active : DATE;
	ostern: DATE;
	i: INT;
	jahr: INT;
	x_date: DATE;
	wday : INT;
END_VAR

(*
version 1.3	24 nov 2007
programmer 	hugo
tested by		tobias

holiday calculates if a given day is a holiday and displays the name of the holiday as string as well as a boolean flag to indicate a holiday.
the holidays can be specified in an array in the constants section of the function block.
a holiday can be of fixed date for example new years day on january 1st.
a holiday can have a fixed offset from easter sunday as for most church holidays.
a holiday can be a specific weekday before a fixed date, for example buss und bettag is the last wednesday before nov 23rd.
with a simple f_use flag any specific holiday can be turned on or off if needed.
The setup Variables Friday, Saturday and Sunday can be used to activate the output on the specific weekday.

*)
(* for performance reasons only activate once a day *)
IF last_active = date_in THEN RETURN; END_IF;

(* berechnung von ostern für das aktuelle jahr *)
jahr := year(date_in);
Ostern := easter(jahr);
last_active := Date_in;

